REGION Network 40: MGF BACKWASH INLET VALVE ABFV-103 OPEN COMMOND FAIL
   RUNG wire#powerrail
      Contact( "FLUSH DB"."ABFV 103 MULTIGRADE FILTER VALVE" )
      wire#w1
      Coil( "ALARM DB"."MGF BACKWASH INLET VALVE ABFV-103 OPEN COMMOND FAIL" )
   END_RUNG
   RUNG wire#w1
      P_Trig( "P_TRIG".ARR[39] )
      S_Coil( "OUTPUT MAPPING DB"."HOOTER RESET" )
   END_RUNG
   // the same network as SCL:
   "ALARM DB"."MGF BACKWASH INLET VALVE ABFV-103 OPEN COMMOND FAIL" := "FLUSH DB"."ABFV 103 MULTIGRADE FILTER VALVE";
   #_w1 := "FLUSH DB"."ABFV 103 MULTIGRADE FILTER VALVE" AND NOT "P_TRIG".ARR[39];   // rising edge
   "P_TRIG".ARR[39] := "FLUSH DB"."ABFV 103 MULTIGRADE FILTER VALVE";
   IF #_w1 THEN "OUTPUT MAPPING DB"."HOOTER RESET" := TRUE; END_IF;
END_REGION

REGION Network 41: MGF BACKWASH INLET VALVE ABFV-103 CLOSE COMMOND FAIL
   RUNG wire#powerrail
      Contact( "FLUSH DB"."ABFV 103 MULTIGRADE FILTER VALVE_CLOSE" )
      wire#w1
      Coil( "ALARM DB"."MGF BACKWASH INLET VALVE ABFV-103 CLOSE COMMOND FAIL" )
   END_RUNG
   RUNG wire#w1
      P_Trig( "P_TRIG".ARR[40] )
      S_Coil( "OUTPUT MAPPING DB"."HOOTER RESET" )
   END_RUNG
   // the same network as SCL:
   "ALARM DB"."MGF BACKWASH INLET VALVE ABFV-103 CLOSE COMMOND FAIL" := "FLUSH DB"."ABFV 103 MULTIGRADE FILTER VALVE_CLOSE";
   #_w1 := "FLUSH DB"."ABFV 103 MULTIGRADE FILTER VALVE_CLOSE" AND NOT "P_TRIG".ARR[40];   // rising edge
   "P_TRIG".ARR[40] := "FLUSH DB"."ABFV 103 MULTIGRADE FILTER VALVE_CLOSE";
   IF #_w1 THEN "OUTPUT MAPPING DB"."HOOTER RESET" := TRUE; END_IF;
END_REGION

REGION Network 42: MGF OUTLET VALVE ABFV-104 OPEN COMMOND FAIL
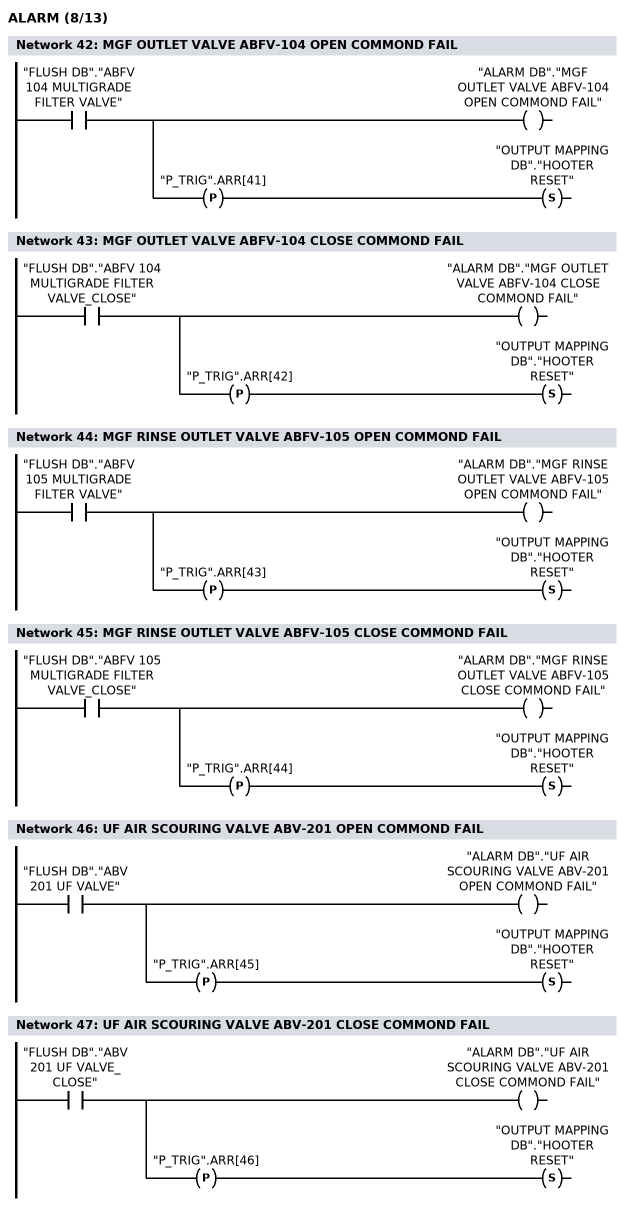
   RUNG wire#powerrail
      Contact( "FLUSH DB"."ABFV 104 MULTIGRADE FILTER VALVE" )
      wire#w1
      Coil( "ALARM DB"."MGF OUTLET VALVE ABFV-104 OPEN COMMOND FAIL" )
   END_RUNG
   RUNG wire#w1
      P_Trig( "P_TRIG".ARR[41] )
      S_Coil( "OUTPUT MAPPING DB"."HOOTER RESET" )
   END_RUNG
   // the same network as SCL:
   "ALARM DB"."MGF OUTLET VALVE ABFV-104 OPEN COMMOND FAIL" := "FLUSH DB"."ABFV 104 MULTIGRADE FILTER VALVE";
   #_w1 := "FLUSH DB"."ABFV 104 MULTIGRADE FILTER VALVE" AND NOT "P_TRIG".ARR[41];   // rising edge
   "P_TRIG".ARR[41] := "FLUSH DB"."ABFV 104 MULTIGRADE FILTER VALVE";
   IF #_w1 THEN "OUTPUT MAPPING DB"."HOOTER RESET" := TRUE; END_IF;
END_REGION

REGION Network 43: MGF OUTLET VALVE ABFV-104 CLOSE COMMOND FAIL
   RUNG wire#powerrail
      Contact( "FLUSH DB"."ABFV 104 MULTIGRADE FILTER VALVE_CLOSE" )
      wire#w1
      Coil( "ALARM DB"."MGF OUTLET VALVE ABFV-104 CLOSE COMMOND FAIL" )
   END_RUNG
   RUNG wire#w1
      P_Trig( "P_TRIG".ARR[42] )
      S_Coil( "OUTPUT MAPPING DB"."HOOTER RESET" )
   END_RUNG
   // the same network as SCL:
   "ALARM DB"."MGF OUTLET VALVE ABFV-104 CLOSE COMMOND FAIL" := "FLUSH DB"."ABFV 104 MULTIGRADE FILTER VALVE_CLOSE";
   #_w1 := "FLUSH DB"."ABFV 104 MULTIGRADE FILTER VALVE_CLOSE" AND NOT "P_TRIG".ARR[42];   // rising edge
   "P_TRIG".ARR[42] := "FLUSH DB"."ABFV 104 MULTIGRADE FILTER VALVE_CLOSE";
   IF #_w1 THEN "OUTPUT MAPPING DB"."HOOTER RESET" := TRUE; END_IF;
END_REGION

REGION Network 44: MGF RINSE OUTLET VALVE ABFV-105 OPEN COMMOND FAIL
   RUNG wire#powerrail
      Contact( "FLUSH DB"."ABFV 105 MULTIGRADE FILTER VALVE" )
      wire#w1
      Coil( "ALARM DB"."MGF RINSE OUTLET VALVE ABFV-105 OPEN COMMOND FAIL" )
   END_RUNG
   RUNG wire#w1
      P_Trig( "P_TRIG".ARR[43] )
      S_Coil( "OUTPUT MAPPING DB"."HOOTER RESET" )
   END_RUNG
   // the same network as SCL:
   "ALARM DB"."MGF RINSE OUTLET VALVE ABFV-105 OPEN COMMOND FAIL" := "FLUSH DB"."ABFV 105 MULTIGRADE FILTER VALVE";
   #_w1 := "FLUSH DB"."ABFV 105 MULTIGRADE FILTER VALVE" AND NOT "P_TRIG".ARR[43];   // rising edge
   "P_TRIG".ARR[43] := "FLUSH DB"."ABFV 105 MULTIGRADE FILTER VALVE";
   IF #_w1 THEN "OUTPUT MAPPING DB"."HOOTER RESET" := TRUE; END_IF;
END_REGION

REGION Network 45: MGF RINSE OUTLET VALVE ABFV-105 CLOSE COMMOND FAIL
   RUNG wire#powerrail
      Contact( "FLUSH DB"."ABFV 105 MULTIGRADE FILTER VALVE_CLOSE" )
      wire#w1
      Coil( "ALARM DB"."MGF RINSE OUTLET VALVE ABFV-105 CLOSE COMMOND FAIL" )
   END_RUNG
   RUNG wire#w1
      P_Trig( "P_TRIG".ARR[44] )
      S_Coil( "OUTPUT MAPPING DB"."HOOTER RESET" )
   END_RUNG
   // the same network as SCL:
   "ALARM DB"."MGF RINSE OUTLET VALVE ABFV-105 CLOSE COMMOND FAIL" := "FLUSH DB"."ABFV 105 MULTIGRADE FILTER VALVE_CLOSE";
   #_w1 := "FLUSH DB"."ABFV 105 MULTIGRADE FILTER VALVE_CLOSE" AND NOT "P_TRIG".ARR[44];   // rising edge
   "P_TRIG".ARR[44] := "FLUSH DB"."ABFV 105 MULTIGRADE FILTER VALVE_CLOSE";
   IF #_w1 THEN "OUTPUT MAPPING DB"."HOOTER RESET" := TRUE; END_IF;
END_REGION

REGION Network 46: UF AIR SCOURING VALVE ABV-201 OPEN COMMOND FAIL
   RUNG wire#powerrail
      Contact( "FLUSH DB"."ABV 201 UF VALVE" )
      wire#w1
      Coil( "ALARM DB"."UF AIR SCOURING VALVE ABV-201 OPEN COMMOND FAIL" )
   END_RUNG
   RUNG wire#w1
      P_Trig( "P_TRIG".ARR[45] )
      S_Coil( "OUTPUT MAPPING DB"."HOOTER RESET" )
   END_RUNG
   // the same network as SCL:
   "ALARM DB"."UF AIR SCOURING VALVE ABV-201 OPEN COMMOND FAIL" := "FLUSH DB"."ABV 201 UF VALVE";
   #_w1 := "FLUSH DB"."ABV 201 UF VALVE" AND NOT "P_TRIG".ARR[45];   // rising edge
   "P_TRIG".ARR[45] := "FLUSH DB"."ABV 201 UF VALVE";
   IF #_w1 THEN "OUTPUT MAPPING DB"."HOOTER RESET" := TRUE; END_IF;
END_REGION

REGION Network 47: UF AIR SCOURING VALVE ABV-201 CLOSE COMMOND FAIL
   RUNG wire#powerrail
      Contact( "FLUSH DB"."ABV 201 UF VALVE_CLOSE" )
      wire#w1
      Coil( "ALARM DB"."UF AIR SCOURING VALVE ABV-201 CLOSE COMMOND FAIL" )
   END_RUNG
   RUNG wire#w1
      P_Trig( "P_TRIG".ARR[46] )
      S_Coil( "OUTPUT MAPPING DB"."HOOTER RESET" )
   END_RUNG
   // the same network as SCL:
   "ALARM DB"."UF AIR SCOURING VALVE ABV-201 CLOSE COMMOND FAIL" := "FLUSH DB"."ABV 201 UF VALVE_CLOSE";
   #_w1 := "FLUSH DB"."ABV 201 UF VALVE_CLOSE" AND NOT "P_TRIG".ARR[46];   // rising edge
   "P_TRIG".ARR[46] := "FLUSH DB"."ABV 201 UF VALVE_CLOSE";
   IF #_w1 THEN "OUTPUT MAPPING DB"."HOOTER RESET" := TRUE; END_IF;
END_REGION

REGION Network 48: UF INLET VALVE ABFV-201 OPEN COMMOND FAIL
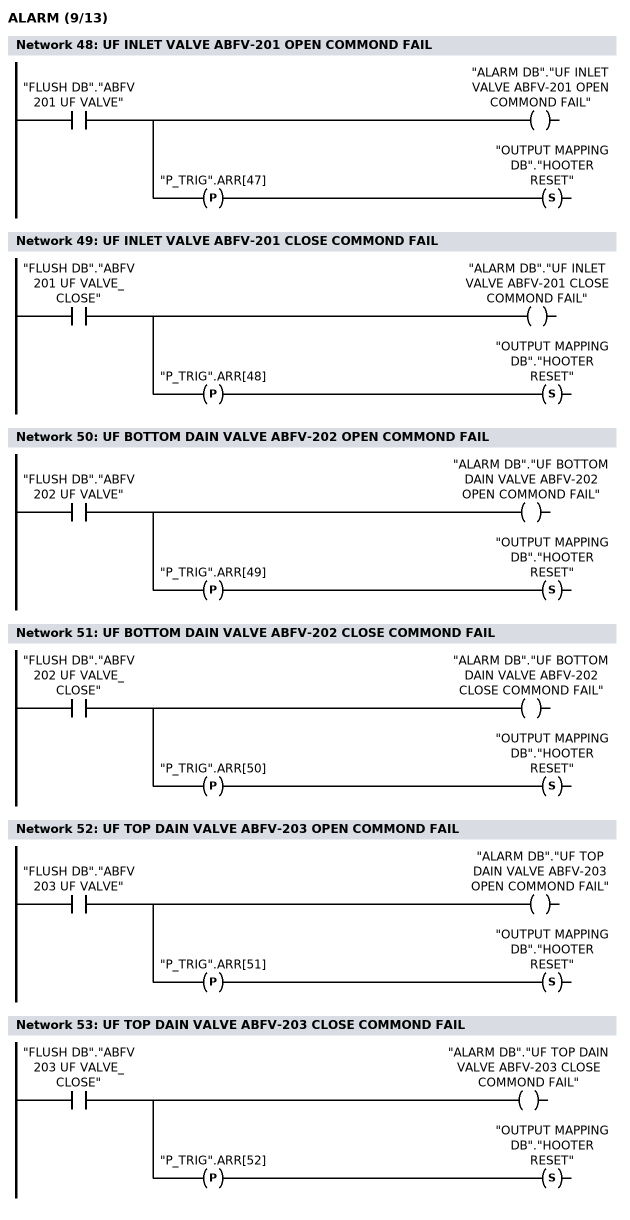
   RUNG wire#powerrail
      Contact( "FLUSH DB"."ABFV 201 UF VALVE" )
      wire#w1
      Coil( "ALARM DB"."UF INLET VALVE ABFV-201 OPEN COMMOND FAIL" )
   END_RUNG
   RUNG wire#w1
      P_Trig( "P_TRIG".ARR[47] )
      S_Coil( "OUTPUT MAPPING DB"."HOOTER RESET" )
   END_RUNG
   // the same network as SCL:
   "ALARM DB"."UF INLET VALVE ABFV-201 OPEN COMMOND FAIL" := "FLUSH DB"."ABFV 201 UF VALVE";
   #_w1 := "FLUSH DB"."ABFV 201 UF VALVE" AND NOT "P_TRIG".ARR[47];   // rising edge
   "P_TRIG".ARR[47] := "FLUSH DB"."ABFV 201 UF VALVE";
   IF #_w1 THEN "OUTPUT MAPPING DB"."HOOTER RESET" := TRUE; END_IF;
END_REGION

REGION Network 49: UF INLET VALVE ABFV-201 CLOSE COMMOND FAIL
   RUNG wire#powerrail
      Contact( "FLUSH DB"."ABFV 201 UF VALVE_CLOSE" )
      wire#w1
      Coil( "ALARM DB"."UF INLET VALVE ABFV-201 CLOSE COMMOND FAIL" )
   END_RUNG
   RUNG wire#w1
      P_Trig( "P_TRIG".ARR[48] )
      S_Coil( "OUTPUT MAPPING DB"."HOOTER RESET" )
   END_RUNG
   // the same network as SCL:
   "ALARM DB"."UF INLET VALVE ABFV-201 CLOSE COMMOND FAIL" := "FLUSH DB"."ABFV 201 UF VALVE_CLOSE";
   #_w1 := "FLUSH DB"."ABFV 201 UF VALVE_CLOSE" AND NOT "P_TRIG".ARR[48];   // rising edge
   "P_TRIG".ARR[48] := "FLUSH DB"."ABFV 201 UF VALVE_CLOSE";
   IF #_w1 THEN "OUTPUT MAPPING DB"."HOOTER RESET" := TRUE; END_IF;
END_REGION

REGION Network 50: UF BOTTOM DAIN VALVE ABFV-202 OPEN COMMOND FAIL
   RUNG wire#powerrail
      Contact( "FLUSH DB"."ABFV 202 UF VALVE" )
      wire#w1
      Coil( "ALARM DB"."UF BOTTOM DAIN VALVE ABFV-202 OPEN COMMOND FAIL" )
   END_RUNG
   RUNG wire#w1
      P_Trig( "P_TRIG".ARR[49] )
      S_Coil( "OUTPUT MAPPING DB"."HOOTER RESET" )
   END_RUNG
   // the same network as SCL:
   "ALARM DB"."UF BOTTOM DAIN VALVE ABFV-202 OPEN COMMOND FAIL" := "FLUSH DB"."ABFV 202 UF VALVE";
   #_w1 := "FLUSH DB"."ABFV 202 UF VALVE" AND NOT "P_TRIG".ARR[49];   // rising edge
   "P_TRIG".ARR[49] := "FLUSH DB"."ABFV 202 UF VALVE";
   IF #_w1 THEN "OUTPUT MAPPING DB"."HOOTER RESET" := TRUE; END_IF;
END_REGION

REGION Network 51: UF BOTTOM DAIN VALVE ABFV-202 CLOSE COMMOND FAIL
   RUNG wire#powerrail
      Contact( "FLUSH DB"."ABFV 202 UF VALVE_CLOSE" )
      wire#w1
      Coil( "ALARM DB"."UF BOTTOM DAIN VALVE ABFV-202 CLOSE COMMOND FAIL" )
   END_RUNG
   RUNG wire#w1
      P_Trig( "P_TRIG".ARR[50] )
      S_Coil( "OUTPUT MAPPING DB"."HOOTER RESET" )
   END_RUNG
   // the same network as SCL:
   "ALARM DB"."UF BOTTOM DAIN VALVE ABFV-202 CLOSE COMMOND FAIL" := "FLUSH DB"."ABFV 202 UF VALVE_CLOSE";
   #_w1 := "FLUSH DB"."ABFV 202 UF VALVE_CLOSE" AND NOT "P_TRIG".ARR[50];   // rising edge
   "P_TRIG".ARR[50] := "FLUSH DB"."ABFV 202 UF VALVE_CLOSE";
   IF #_w1 THEN "OUTPUT MAPPING DB"."HOOTER RESET" := TRUE; END_IF;
END_REGION

REGION Network 52: UF TOP DAIN VALVE ABFV-203 OPEN COMMOND FAIL
   RUNG wire#powerrail
      Contact( "FLUSH DB"."ABFV 203 UF VALVE" )
      wire#w1
      Coil( "ALARM DB"."UF TOP DAIN VALVE ABFV-203 OPEN COMMOND FAIL" )
   END_RUNG
   RUNG wire#w1
      P_Trig( "P_TRIG".ARR[51] )
      S_Coil( "OUTPUT MAPPING DB"."HOOTER RESET" )
   END_RUNG
   // the same network as SCL:
   "ALARM DB"."UF TOP DAIN VALVE ABFV-203 OPEN COMMOND FAIL" := "FLUSH DB"."ABFV 203 UF VALVE";
   #_w1 := "FLUSH DB"."ABFV 203 UF VALVE" AND NOT "P_TRIG".ARR[51];   // rising edge
   "P_TRIG".ARR[51] := "FLUSH DB"."ABFV 203 UF VALVE";
   IF #_w1 THEN "OUTPUT MAPPING DB"."HOOTER RESET" := TRUE; END_IF;
END_REGION

REGION Network 53: UF TOP DAIN VALVE ABFV-203 CLOSE COMMOND FAIL
   RUNG wire#powerrail
      Contact( "FLUSH DB"."ABFV 203 UF VALVE_CLOSE" )
      wire#w1
      Coil( "ALARM DB"."UF TOP DAIN VALVE ABFV-203 CLOSE COMMOND FAIL" )
   END_RUNG
   RUNG wire#w1
      P_Trig( "P_TRIG".ARR[52] )
      S_Coil( "OUTPUT MAPPING DB"."HOOTER RESET" )
   END_RUNG
   // the same network as SCL:
   "ALARM DB"."UF TOP DAIN VALVE ABFV-203 CLOSE COMMOND FAIL" := "FLUSH DB"."ABFV 203 UF VALVE_CLOSE";
   #_w1 := "FLUSH DB"."ABFV 203 UF VALVE_CLOSE" AND NOT "P_TRIG".ARR[52];   // rising edge
   "P_TRIG".ARR[52] := "FLUSH DB"."ABFV 203 UF VALVE_CLOSE";
   IF #_w1 THEN "OUTPUT MAPPING DB"."HOOTER RESET" := TRUE; END_IF;
END_REGION

REGION Network 54: UF BACKWASH INLET VALVE ABFV-204 OPEN COMMOND FAIL
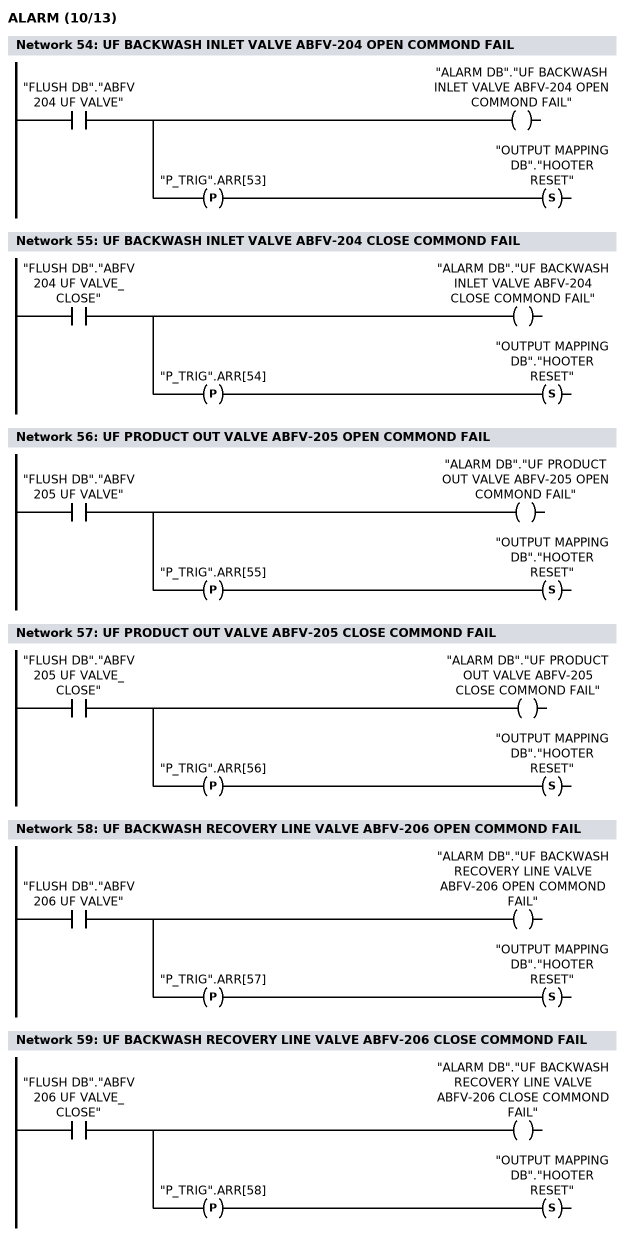
   RUNG wire#powerrail
      Contact( "FLUSH DB"."ABFV 204 UF VALVE" )
      wire#w1
      Coil( "ALARM DB"."UF BACKWASH INLET VALVE ABFV-204 OPEN COMMOND FAIL" )
   END_RUNG
   RUNG wire#w1
      P_Trig( "P_TRIG".ARR[53] )
      S_Coil( "OUTPUT MAPPING DB"."HOOTER RESET" )
   END_RUNG
   // the same network as SCL:
   "ALARM DB"."UF BACKWASH INLET VALVE ABFV-204 OPEN COMMOND FAIL" := "FLUSH DB"."ABFV 204 UF VALVE";
   #_w1 := "FLUSH DB"."ABFV 204 UF VALVE" AND NOT "P_TRIG".ARR[53];   // rising edge
   "P_TRIG".ARR[53] := "FLUSH DB"."ABFV 204 UF VALVE";
   IF #_w1 THEN "OUTPUT MAPPING DB"."HOOTER RESET" := TRUE; END_IF;
END_REGION

REGION Network 55: UF BACKWASH INLET VALVE ABFV-204 CLOSE COMMOND FAIL
   RUNG wire#powerrail
      Contact( "FLUSH DB"."ABFV 204 UF VALVE_CLOSE" )
      wire#w1
      Coil( "ALARM DB"."UF BACKWASH INLET VALVE ABFV-204 CLOSE COMMOND FAIL" )
   END_RUNG
   RUNG wire#w1
      P_Trig( "P_TRIG".ARR[54] )
      S_Coil( "OUTPUT MAPPING DB"."HOOTER RESET" )
   END_RUNG
   // the same network as SCL:
   "ALARM DB"."UF BACKWASH INLET VALVE ABFV-204 CLOSE COMMOND FAIL" := "FLUSH DB"."ABFV 204 UF VALVE_CLOSE";
   #_w1 := "FLUSH DB"."ABFV 204 UF VALVE_CLOSE" AND NOT "P_TRIG".ARR[54];   // rising edge
   "P_TRIG".ARR[54] := "FLUSH DB"."ABFV 204 UF VALVE_CLOSE";
   IF #_w1 THEN "OUTPUT MAPPING DB"."HOOTER RESET" := TRUE; END_IF;
END_REGION

REGION Network 56: UF PRODUCT OUT VALVE ABFV-205 OPEN COMMOND FAIL
   RUNG wire#powerrail
      Contact( "FLUSH DB"."ABFV 205 UF VALVE" )
      wire#w1
      Coil( "ALARM DB"."UF PRODUCT OUT VALVE ABFV-205 OPEN COMMOND FAIL" )
   END_RUNG
   RUNG wire#w1
      P_Trig( "P_TRIG".ARR[55] )
      S_Coil( "OUTPUT MAPPING DB"."HOOTER RESET" )
   END_RUNG
   // the same network as SCL:
   "ALARM DB"."UF PRODUCT OUT VALVE ABFV-205 OPEN COMMOND FAIL" := "FLUSH DB"."ABFV 205 UF VALVE";
   #_w1 := "FLUSH DB"."ABFV 205 UF VALVE" AND NOT "P_TRIG".ARR[55];   // rising edge
   "P_TRIG".ARR[55] := "FLUSH DB"."ABFV 205 UF VALVE";
   IF #_w1 THEN "OUTPUT MAPPING DB"."HOOTER RESET" := TRUE; END_IF;
END_REGION

REGION Network 57: UF PRODUCT OUT VALVE ABFV-205 CLOSE COMMOND FAIL
   RUNG wire#powerrail
      Contact( "FLUSH DB"."ABFV 205 UF VALVE_CLOSE" )
      wire#w1
      Coil( "ALARM DB"."UF PRODUCT OUT VALVE ABFV-205 CLOSE COMMOND FAIL" )
   END_RUNG
   RUNG wire#w1
      P_Trig( "P_TRIG".ARR[56] )
      S_Coil( "OUTPUT MAPPING DB"."HOOTER RESET" )
   END_RUNG
   // the same network as SCL:
   "ALARM DB"."UF PRODUCT OUT VALVE ABFV-205 CLOSE COMMOND FAIL" := "FLUSH DB"."ABFV 205 UF VALVE_CLOSE";
   #_w1 := "FLUSH DB"."ABFV 205 UF VALVE_CLOSE" AND NOT "P_TRIG".ARR[56];   // rising edge
   "P_TRIG".ARR[56] := "FLUSH DB"."ABFV 205 UF VALVE_CLOSE";
   IF #_w1 THEN "OUTPUT MAPPING DB"."HOOTER RESET" := TRUE; END_IF;
END_REGION

REGION Network 58: UF BACKWASH RECOVERY LINE VALVE ABFV-206 OPEN COMMOND FAIL
   RUNG wire#powerrail
      Contact( "FLUSH DB"."ABFV 206 UF VALVE" )
      wire#w1
      Coil( "ALARM DB"."UF BACKWASH RECOVERY LINE VALVE ABFV-206 OPEN COMMOND FAIL" )
   END_RUNG
   RUNG wire#w1
      P_Trig( "P_TRIG".ARR[57] )
      S_Coil( "OUTPUT MAPPING DB"."HOOTER RESET" )
   END_RUNG
   // the same network as SCL:
   "ALARM DB"."UF BACKWASH RECOVERY LINE VALVE ABFV-206 OPEN COMMOND FAIL" := "FLUSH DB"."ABFV 206 UF VALVE";
   #_w1 := "FLUSH DB"."ABFV 206 UF VALVE" AND NOT "P_TRIG".ARR[57];   // rising edge
   "P_TRIG".ARR[57] := "FLUSH DB"."ABFV 206 UF VALVE";
   IF #_w1 THEN "OUTPUT MAPPING DB"."HOOTER RESET" := TRUE; END_IF;
END_REGION

REGION Network 59: UF BACKWASH RECOVERY LINE VALVE ABFV-206 CLOSE COMMOND FAIL
   RUNG wire#powerrail
      Contact( "FLUSH DB"."ABFV 206 UF VALVE_CLOSE" )
      wire#w1
      Coil( "ALARM DB"."UF BACKWASH RECOVERY LINE VALVE ABFV-206 CLOSE COMMOND FAIL" )
   END_RUNG
   RUNG wire#w1
      P_Trig( "P_TRIG".ARR[58] )
      S_Coil( "OUTPUT MAPPING DB"."HOOTER RESET" )
   END_RUNG
   // the same network as SCL:
   "ALARM DB"."UF BACKWASH RECOVERY LINE VALVE ABFV-206 CLOSE COMMOND FAIL" := "FLUSH DB"."ABFV 206 UF VALVE_CLOSE";
   #_w1 := "FLUSH DB"."ABFV 206 UF VALVE_CLOSE" AND NOT "P_TRIG".ARR[58];   // rising edge
   "P_TRIG".ARR[58] := "FLUSH DB"."ABFV 206 UF VALVE_CLOSE";
   IF #_w1 THEN "OUTPUT MAPPING DB"."HOOTER RESET" := TRUE; END_IF;
END_REGION

REGION Network 60: UF BACKWASH DRAIN LINE VALVE ABFV-207 OPEN COMMOND FAIL
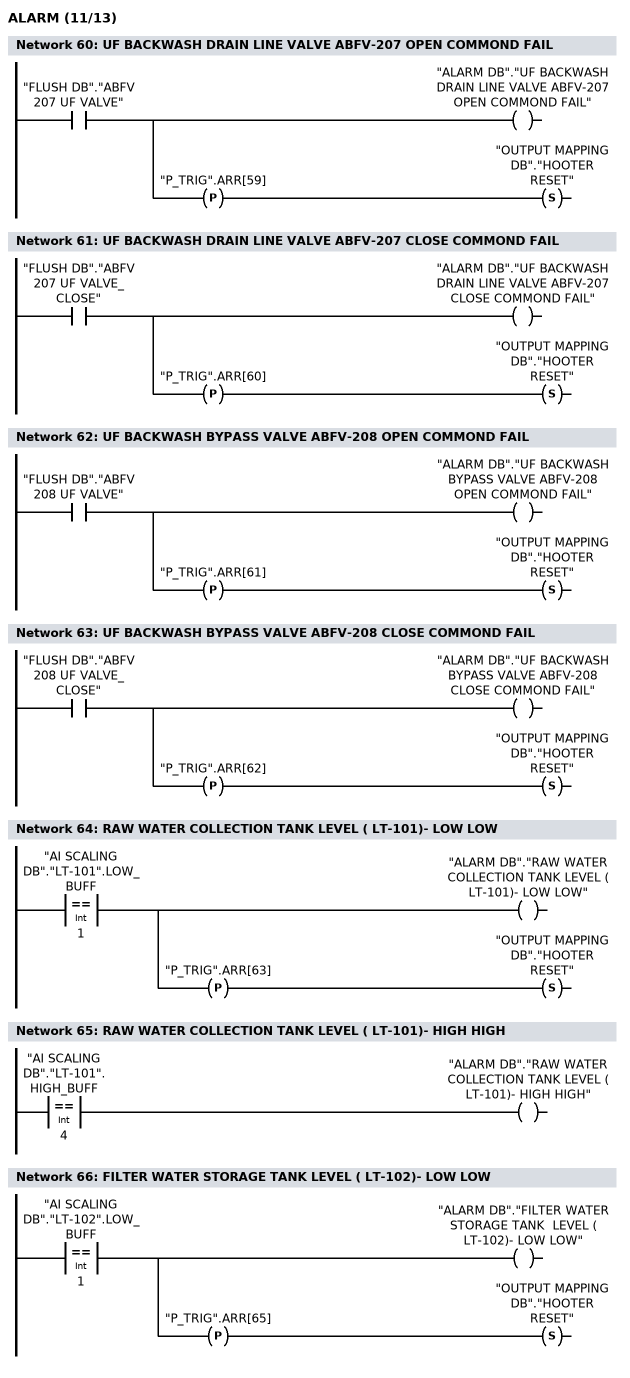
   RUNG wire#powerrail
      Contact( "FLUSH DB"."ABFV 207 UF VALVE" )
      wire#w1
      Coil( "ALARM DB"."UF BACKWASH DRAIN LINE VALVE ABFV-207 OPEN COMMOND FAIL" )
   END_RUNG
   RUNG wire#w1
      P_Trig( "P_TRIG".ARR[59] )
      S_Coil( "OUTPUT MAPPING DB"."HOOTER RESET" )
   END_RUNG
   // the same network as SCL:
   "ALARM DB"."UF BACKWASH DRAIN LINE VALVE ABFV-207 OPEN COMMOND FAIL" := "FLUSH DB"."ABFV 207 UF VALVE";
   #_w1 := "FLUSH DB"."ABFV 207 UF VALVE" AND NOT "P_TRIG".ARR[59];   // rising edge
   "P_TRIG".ARR[59] := "FLUSH DB"."ABFV 207 UF VALVE";
   IF #_w1 THEN "OUTPUT MAPPING DB"."HOOTER RESET" := TRUE; END_IF;
END_REGION

REGION Network 61: UF BACKWASH DRAIN LINE VALVE ABFV-207 CLOSE COMMOND FAIL
   RUNG wire#powerrail
      Contact( "FLUSH DB"."ABFV 207 UF VALVE_CLOSE" )
      wire#w1
      Coil( "ALARM DB"."UF BACKWASH DRAIN LINE VALVE ABFV-207 CLOSE COMMOND FAIL" )
   END_RUNG
   RUNG wire#w1
      P_Trig( "P_TRIG".ARR[60] )
      S_Coil( "OUTPUT MAPPING DB"."HOOTER RESET" )
   END_RUNG
   // the same network as SCL:
   "ALARM DB"."UF BACKWASH DRAIN LINE VALVE ABFV-207 CLOSE COMMOND FAIL" := "FLUSH DB"."ABFV 207 UF VALVE_CLOSE";
   #_w1 := "FLUSH DB"."ABFV 207 UF VALVE_CLOSE" AND NOT "P_TRIG".ARR[60];   // rising edge
   "P_TRIG".ARR[60] := "FLUSH DB"."ABFV 207 UF VALVE_CLOSE";
   IF #_w1 THEN "OUTPUT MAPPING DB"."HOOTER RESET" := TRUE; END_IF;
END_REGION

REGION Network 62: UF BACKWASH BYPASS VALVE ABFV-208 OPEN COMMOND FAIL
   RUNG wire#powerrail
      Contact( "FLUSH DB"."ABFV 208 UF VALVE" )
      wire#w1
      Coil( "ALARM DB"."UF BACKWASH BYPASS VALVE ABFV-208 OPEN COMMOND FAIL" )
   END_RUNG
   RUNG wire#w1
      P_Trig( "P_TRIG".ARR[61] )
      S_Coil( "OUTPUT MAPPING DB"."HOOTER RESET" )
   END_RUNG
   // the same network as SCL:
   "ALARM DB"."UF BACKWASH BYPASS VALVE ABFV-208 OPEN COMMOND FAIL" := "FLUSH DB"."ABFV 208 UF VALVE";
   #_w1 := "FLUSH DB"."ABFV 208 UF VALVE" AND NOT "P_TRIG".ARR[61];   // rising edge
   "P_TRIG".ARR[61] := "FLUSH DB"."ABFV 208 UF VALVE";
   IF #_w1 THEN "OUTPUT MAPPING DB"."HOOTER RESET" := TRUE; END_IF;
END_REGION

REGION Network 63: UF BACKWASH BYPASS VALVE ABFV-208 CLOSE COMMOND FAIL
   RUNG wire#powerrail
      Contact( "FLUSH DB"."ABFV 208 UF VALVE_CLOSE" )
      wire#w1
      Coil( "ALARM DB"."UF BACKWASH BYPASS VALVE ABFV-208 CLOSE COMMOND FAIL" )
   END_RUNG
   RUNG wire#w1
      P_Trig( "P_TRIG".ARR[62] )
      S_Coil( "OUTPUT MAPPING DB"."HOOTER RESET" )
   END_RUNG
   // the same network as SCL:
   "ALARM DB"."UF BACKWASH BYPASS VALVE ABFV-208 CLOSE COMMOND FAIL" := "FLUSH DB"."ABFV 208 UF VALVE_CLOSE";
   #_w1 := "FLUSH DB"."ABFV 208 UF VALVE_CLOSE" AND NOT "P_TRIG".ARR[62];   // rising edge
   "P_TRIG".ARR[62] := "FLUSH DB"."ABFV 208 UF VALVE_CLOSE";
   IF #_w1 THEN "OUTPUT MAPPING DB"."HOOTER RESET" := TRUE; END_IF;
END_REGION

REGION Network 64: RAW WATER COLLECTION TANK LEVEL ( LT-101)- LOW LOW
   RUNG wire#powerrail
      { S7_Templates := "SrcType := Int" } EQ_Contact(in1 := "AI SCALING DB"."LT-101".LOW_BUFF, in2 := 1)
      wire#w1
      Coil( "ALARM DB"."RAW WATER COLLECTION TANK LEVEL ( LT-101)- LOW LOW" )
   END_RUNG
   RUNG wire#w1
      P_Trig( "P_TRIG".ARR[63] )
      S_Coil( "OUTPUT MAPPING DB"."HOOTER RESET" )
   END_RUNG
   // the same network as SCL:
   "ALARM DB"."RAW WATER COLLECTION TANK LEVEL ( LT-101)- LOW LOW" := "AI SCALING DB"."LT-101".LOW_BUFF = 1;
   #_w1 := "ALARM DB"."RAW WATER COLLECTION TANK LEVEL ( LT-101)- LOW LOW" AND NOT "P_TRIG".ARR[63];   // rising edge
   "P_TRIG".ARR[63] := "ALARM DB"."RAW WATER COLLECTION TANK LEVEL ( LT-101)- LOW LOW";
   IF #_w1 THEN "OUTPUT MAPPING DB"."HOOTER RESET" := TRUE; END_IF;
END_REGION

REGION Network 65: RAW WATER COLLECTION TANK LEVEL ( LT-101)- HIGH HIGH
   RUNG wire#powerrail
      { S7_Templates := "SrcType := Int" } EQ_Contact(in1 := "AI SCALING DB"."LT-101".HIGH_BUFF, in2 := 4)
      Coil( "ALARM DB"."RAW WATER COLLECTION TANK LEVEL ( LT-101)- HIGH HIGH" )
   END_RUNG
   // the same network as SCL:
   "ALARM DB"."RAW WATER COLLECTION TANK LEVEL ( LT-101)- HIGH HIGH" := "AI SCALING DB"."LT-101".HIGH_BUFF = 4;
END_REGION

REGION Network 66: FILTER WATER STORAGE TANK LEVEL ( LT-102)- LOW LOW
   RUNG wire#powerrail
      { S7_Templates := "SrcType := Int" } EQ_Contact(in1 := "AI SCALING DB"."LT-102".LOW_BUFF, in2 := 1)
      wire#w1
      Coil( "ALARM DB"."FILTER WATER STORAGE TANK  LEVEL ( LT-102)- LOW LOW" )
   END_RUNG
   RUNG wire#w1
      P_Trig( "P_TRIG".ARR[65] )
      S_Coil( "OUTPUT MAPPING DB"."HOOTER RESET" )
   END_RUNG
   // the same network as SCL:
   "ALARM DB"."FILTER WATER STORAGE TANK  LEVEL ( LT-102)- LOW LOW" := "AI SCALING DB"."LT-102".LOW_BUFF = 1;
   #_w1 := "ALARM DB"."FILTER WATER STORAGE TANK  LEVEL ( LT-102)- LOW LOW" AND NOT "P_TRIG".ARR[65];   // rising edge
   "P_TRIG".ARR[65] := "ALARM DB"."FILTER WATER STORAGE TANK  LEVEL ( LT-102)- LOW LOW";
   IF #_w1 THEN "OUTPUT MAPPING DB"."HOOTER RESET" := TRUE; END_IF;
END_REGION

REGION Network 67: FILTER WATER STORAGE TANK LEVEL ( LT-102)- HIGH HIGH
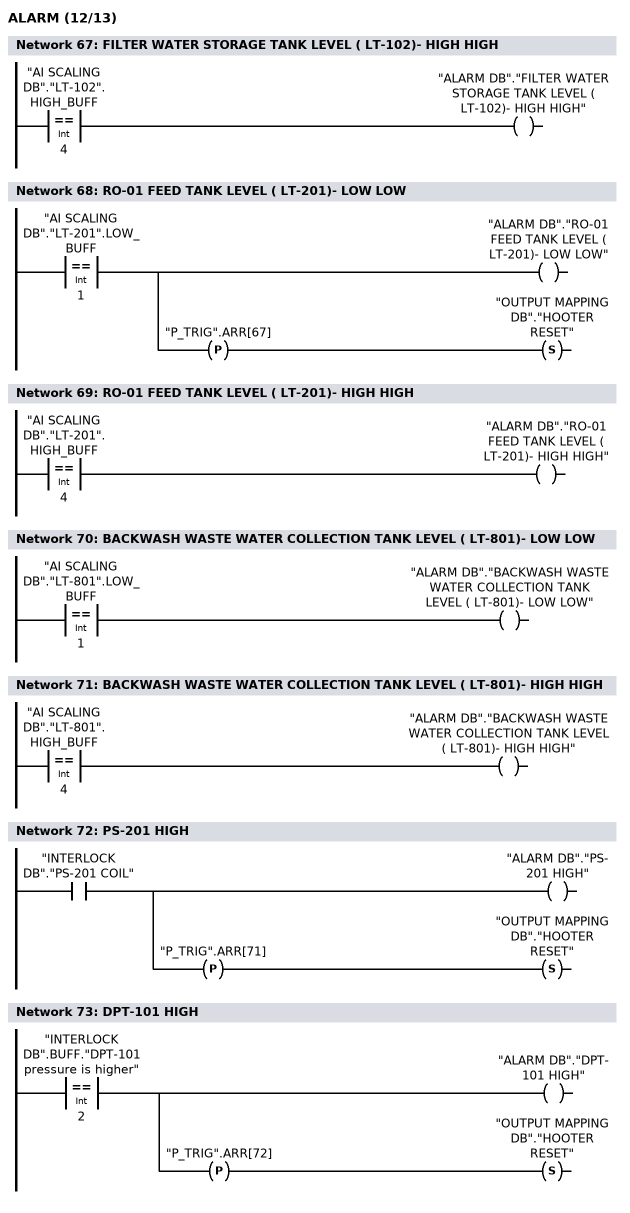
   RUNG wire#powerrail
      { S7_Templates := "SrcType := Int" } EQ_Contact(in1 := "AI SCALING DB"."LT-102".HIGH_BUFF, in2 := 4)
      Coil( "ALARM DB"."FILTER WATER STORAGE TANK LEVEL ( LT-102)- HIGH HIGH" )
   END_RUNG
   // the same network as SCL:
   "ALARM DB"."FILTER WATER STORAGE TANK LEVEL ( LT-102)- HIGH HIGH" := "AI SCALING DB"."LT-102".HIGH_BUFF = 4;
END_REGION

REGION Network 68: RO-01 FEED TANK LEVEL ( LT-201)- LOW LOW
   RUNG wire#powerrail
      { S7_Templates := "SrcType := Int" } EQ_Contact(in1 := "AI SCALING DB"."LT-201".LOW_BUFF, in2 := 1)
      wire#w1
      Coil( "ALARM DB"."RO-01 FEED TANK LEVEL ( LT-201)- LOW LOW" )
   END_RUNG
   RUNG wire#w1
      P_Trig( "P_TRIG".ARR[67] )
      S_Coil( "OUTPUT MAPPING DB"."HOOTER RESET" )
   END_RUNG
   // the same network as SCL:
   "ALARM DB"."RO-01 FEED TANK LEVEL ( LT-201)- LOW LOW" := "AI SCALING DB"."LT-201".LOW_BUFF = 1;
   #_w1 := "ALARM DB"."RO-01 FEED TANK LEVEL ( LT-201)- LOW LOW" AND NOT "P_TRIG".ARR[67];   // rising edge
   "P_TRIG".ARR[67] := "ALARM DB"."RO-01 FEED TANK LEVEL ( LT-201)- LOW LOW";
   IF #_w1 THEN "OUTPUT MAPPING DB"."HOOTER RESET" := TRUE; END_IF;
END_REGION

REGION Network 69: RO-01 FEED TANK LEVEL ( LT-201)- HIGH HIGH
   RUNG wire#powerrail
      { S7_Templates := "SrcType := Int" } EQ_Contact(in1 := "AI SCALING DB"."LT-201".HIGH_BUFF, in2 := 4)
      Coil( "ALARM DB"."RO-01 FEED TANK LEVEL ( LT-201)- HIGH HIGH" )
   END_RUNG
   // the same network as SCL:
   "ALARM DB"."RO-01 FEED TANK LEVEL ( LT-201)- HIGH HIGH" := "AI SCALING DB"."LT-201".HIGH_BUFF = 4;
END_REGION

REGION Network 70: BACKWASH WASTE WATER COLLECTION TANK LEVEL ( LT-801)- LOW LOW
   RUNG wire#powerrail
      { S7_Templates := "SrcType := Int" } EQ_Contact(in1 := "AI SCALING DB"."LT-801".LOW_BUFF, in2 := 1)
      Coil( "ALARM DB"."BACKWASH WASTE WATER COLLECTION TANK  LEVEL ( LT-801)- LOW LOW" )
   END_RUNG
   // the same network as SCL:
   "ALARM DB"."BACKWASH WASTE WATER COLLECTION TANK  LEVEL ( LT-801)- LOW LOW" := "AI SCALING DB"."LT-801".LOW_BUFF = 1;
END_REGION

REGION Network 71: BACKWASH WASTE WATER COLLECTION TANK LEVEL ( LT-801)- HIGH HIGH
   RUNG wire#powerrail
      { S7_Templates := "SrcType := Int" } EQ_Contact(in1 := "AI SCALING DB"."LT-801".HIGH_BUFF, in2 := 4)
      Coil( "ALARM DB"."BACKWASH WASTE WATER COLLECTION TANK LEVEL ( LT-801)- HIGH HIGH" )
   END_RUNG
   // the same network as SCL:
   "ALARM DB"."BACKWASH WASTE WATER COLLECTION TANK LEVEL ( LT-801)- HIGH HIGH" := "AI SCALING DB"."LT-801".HIGH_BUFF = 4;
END_REGION

REGION Network 72: PS-201 HIGH
   RUNG wire#powerrail
      Contact( "INTERLOCK DB"."PS-201 COIL" )
      wire#w1
      Coil( "ALARM DB"."PS-201 HIGH" )
   END_RUNG
   RUNG wire#w1
      P_Trig( "P_TRIG".ARR[71] )
      S_Coil( "OUTPUT MAPPING DB"."HOOTER RESET" )
   END_RUNG
   // the same network as SCL:
   "ALARM DB"."PS-201 HIGH" := "INTERLOCK DB"."PS-201 COIL";
   #_w1 := "INTERLOCK DB"."PS-201 COIL" AND NOT "P_TRIG".ARR[71];   // rising edge
   "P_TRIG".ARR[71] := "INTERLOCK DB"."PS-201 COIL";
   IF #_w1 THEN "OUTPUT MAPPING DB"."HOOTER RESET" := TRUE; END_IF;
END_REGION

REGION Network 73: DPT-101 HIGH
   RUNG wire#powerrail
      { S7_Templates := "SrcType := Int" } EQ_Contact(in1 := "INTERLOCK DB".BUFF."DPT-101 pressure is higher", in2 := 2)
      wire#w1
      Coil( "ALARM DB"."DPT-101 HIGH" )
   END_RUNG
   RUNG wire#w1
      P_Trig( "P_TRIG".ARR[72] )
      S_Coil( "OUTPUT MAPPING DB"."HOOTER RESET" )
   END_RUNG
   // the same network as SCL:
   "ALARM DB"."DPT-101 HIGH" := "INTERLOCK DB".BUFF."DPT-101 pressure is higher" = 2;
   #_w1 := "ALARM DB"."DPT-101 HIGH" AND NOT "P_TRIG".ARR[72];   // rising edge
   "P_TRIG".ARR[72] := "ALARM DB"."DPT-101 HIGH";
   IF #_w1 THEN "OUTPUT MAPPING DB"."HOOTER RESET" := TRUE; END_IF;
END_REGION

REGION Network 74: DPT-201 HIGH
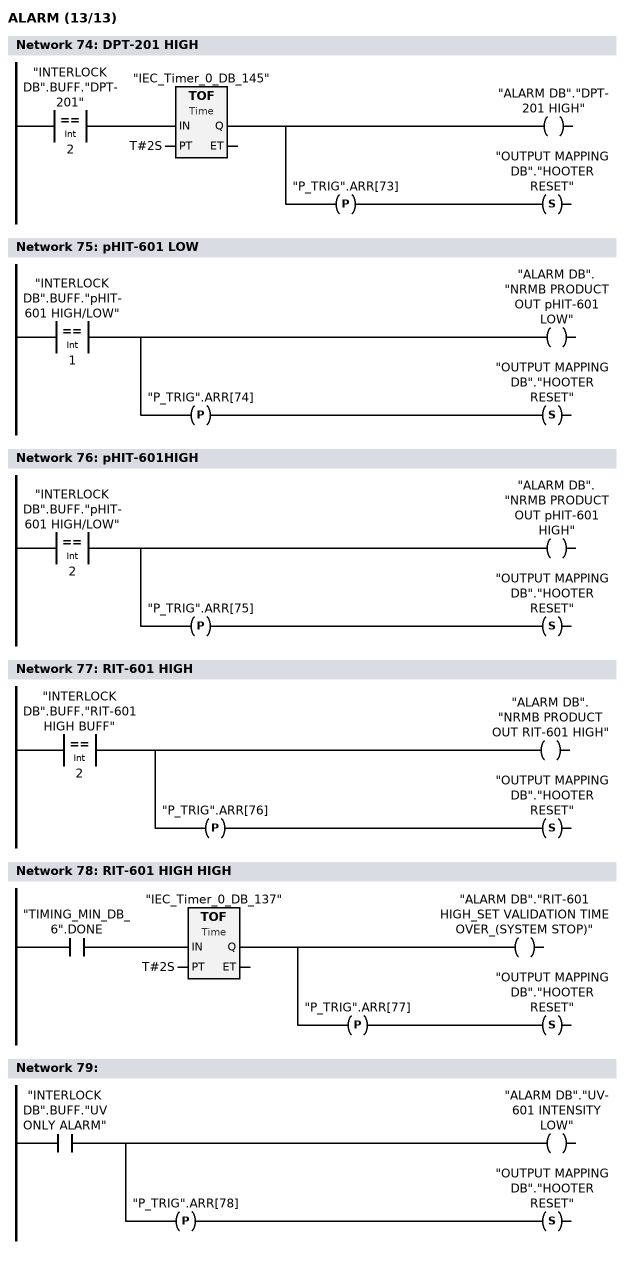
   RUNG wire#powerrail
      { S7_Templates := "SrcType := Int" } EQ_Contact(in1 := "INTERLOCK DB".BUFF."DPT-201", in2 := 2)
      { S7_Templates := "time_type := Time" } "IEC_Timer_0_DB_145".TOF(pt := T#2S, et =>)
      wire#w1
      Coil( "ALARM DB"."DPT-201 HIGH" )
   END_RUNG
   RUNG wire#w1
      P_Trig( "P_TRIG".ARR[73] )
      S_Coil( "OUTPUT MAPPING DB"."HOOTER RESET" )
   END_RUNG
   // the same network as SCL:
   "IEC_Timer_0_DB_145".TOF(IN := "INTERLOCK DB".BUFF."DPT-201" = 2, PT := T#2S);
   "ALARM DB"."DPT-201 HIGH" := "IEC_Timer_0_DB_145".Q;
   #_w1 := "IEC_Timer_0_DB_145".Q AND NOT "P_TRIG".ARR[73];   // rising edge
   "P_TRIG".ARR[73] := "IEC_Timer_0_DB_145".Q;
   IF #_w1 THEN "OUTPUT MAPPING DB"."HOOTER RESET" := TRUE; END_IF;
END_REGION

REGION Network 75: pHIT-601 LOW
   RUNG wire#powerrail
      { S7_Templates := "SrcType := Int" } EQ_Contact(in1 := "INTERLOCK DB".BUFF."pHIT-601 HIGH/LOW", in2 := 1)
      wire#w1
      Coil( "ALARM DB"."NRMB PRODUCT OUT pHIT-601 LOW" )
   END_RUNG
   RUNG wire#w1
      P_Trig( "P_TRIG".ARR[74] )
      S_Coil( "OUTPUT MAPPING DB"."HOOTER RESET" )
   END_RUNG
   // the same network as SCL:
   "ALARM DB"."NRMB PRODUCT OUT pHIT-601 LOW" := "INTERLOCK DB".BUFF."pHIT-601 HIGH/LOW" = 1;
   #_w1 := "ALARM DB"."NRMB PRODUCT OUT pHIT-601 LOW" AND NOT "P_TRIG".ARR[74];   // rising edge
   "P_TRIG".ARR[74] := "ALARM DB"."NRMB PRODUCT OUT pHIT-601 LOW";
   IF #_w1 THEN "OUTPUT MAPPING DB"."HOOTER RESET" := TRUE; END_IF;
END_REGION

REGION Network 76: pHIT-601HIGH
   RUNG wire#powerrail
      { S7_Templates := "SrcType := Int" } EQ_Contact(in1 := "INTERLOCK DB".BUFF."pHIT-601 HIGH/LOW", in2 := 2)
      wire#w1
      Coil( "ALARM DB"."NRMB PRODUCT OUT pHIT-601 HIGH" )
   END_RUNG
   RUNG wire#w1
      P_Trig( "P_TRIG".ARR[75] )
      S_Coil( "OUTPUT MAPPING DB"."HOOTER RESET" )
   END_RUNG
   // the same network as SCL:
   "ALARM DB"."NRMB PRODUCT OUT pHIT-601 HIGH" := "INTERLOCK DB".BUFF."pHIT-601 HIGH/LOW" = 2;
   #_w1 := "ALARM DB"."NRMB PRODUCT OUT pHIT-601 HIGH" AND NOT "P_TRIG".ARR[75];   // rising edge
   "P_TRIG".ARR[75] := "ALARM DB"."NRMB PRODUCT OUT pHIT-601 HIGH";
   IF #_w1 THEN "OUTPUT MAPPING DB"."HOOTER RESET" := TRUE; END_IF;
END_REGION

REGION Network 77: RIT-601 HIGH
   RUNG wire#powerrail
      { S7_Templates := "SrcType := Int" } EQ_Contact(in1 := "INTERLOCK DB".BUFF."RIT-601 HIGH BUFF", in2 := 2)
      wire#w1
      Coil( "ALARM DB"."NRMB PRODUCT OUT RIT-601 HIGH" )
   END_RUNG
   RUNG wire#w1
      P_Trig( "P_TRIG".ARR[76] )
      S_Coil( "OUTPUT MAPPING DB"."HOOTER RESET" )
   END_RUNG
   // the same network as SCL:
   "ALARM DB"."NRMB PRODUCT OUT RIT-601 HIGH" := "INTERLOCK DB".BUFF."RIT-601 HIGH BUFF" = 2;
   #_w1 := "ALARM DB"."NRMB PRODUCT OUT RIT-601 HIGH" AND NOT "P_TRIG".ARR[76];   // rising edge
   "P_TRIG".ARR[76] := "ALARM DB"."NRMB PRODUCT OUT RIT-601 HIGH";
   IF #_w1 THEN "OUTPUT MAPPING DB"."HOOTER RESET" := TRUE; END_IF;
END_REGION

REGION Network 78: RIT-601 HIGH HIGH
   RUNG wire#powerrail
      Contact( "TIMING_MIN_DB_6".DONE )
      { S7_Templates := "time_type := Time" } "IEC_Timer_0_DB_137".TOF(pt := T#2S, et =>)
      wire#w1
      Coil( "ALARM DB"."RIT-601 HIGH_SET VALIDATION TIME OVER_(SYSTEM STOP)" )
   END_RUNG
   RUNG wire#w1
      P_Trig( "P_TRIG".ARR[77] )
      S_Coil( "OUTPUT MAPPING DB"."HOOTER RESET" )
   END_RUNG
   // the same network as SCL:
   "IEC_Timer_0_DB_137".TOF(IN := "TIMING_MIN_DB_6".DONE, PT := T#2S);
   "ALARM DB"."RIT-601 HIGH_SET VALIDATION TIME OVER_(SYSTEM STOP)" := "IEC_Timer_0_DB_137".Q;
   #_w1 := "IEC_Timer_0_DB_137".Q AND NOT "P_TRIG".ARR[77];   // rising edge
   "P_TRIG".ARR[77] := "IEC_Timer_0_DB_137".Q;
   IF #_w1 THEN "OUTPUT MAPPING DB"."HOOTER RESET" := TRUE; END_IF;
END_REGION

REGION Network 79
   RUNG wire#powerrail
      Contact( "INTERLOCK DB".BUFF."UV ONLY ALARM" )
      wire#w1
      Coil( "ALARM DB"."UV-601 INTENSITY LOW" )
   END_RUNG
   RUNG wire#w1
      P_Trig( "P_TRIG".ARR[78] )
      S_Coil( "OUTPUT MAPPING DB"."HOOTER RESET" )
   END_RUNG
   // the same network as SCL:
   "ALARM DB"."UV-601 INTENSITY LOW" := "INTERLOCK DB".BUFF."UV ONLY ALARM";
   #_w1 := "INTERLOCK DB".BUFF."UV ONLY ALARM" AND NOT "P_TRIG".ARR[78];   // rising edge
   "P_TRIG".ARR[78] := "INTERLOCK DB".BUFF."UV ONLY ALARM";
   IF #_w1 THEN "OUTPUT MAPPING DB"."HOOTER RESET" := TRUE; END_IF;
END_REGION
END_FUNCTION

FUNCTION "DATE&TIMES" : Void   // FC9, LAD
{ S7_Optimized_Access := 'TRUE' }
// stored: SetENOAutomatically false
BEGIN

REGION Network 1
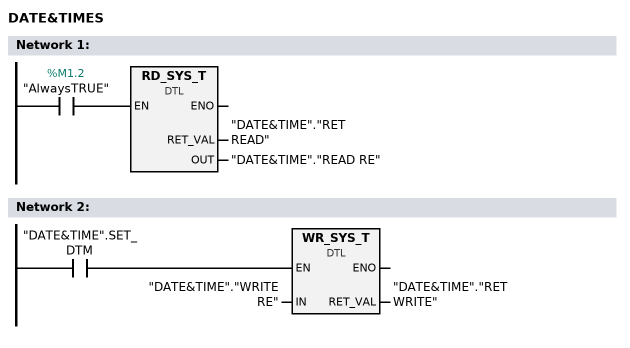
   RUNG wire#powerrail
      Contact( "AlwaysTRUE" )
      { S7_Templates := "date_type := DTL" } RD_SYS_T(RET_VAL => "DATE&TIME"."RET READ", OUT => "DATE&TIME"."READ RE")
   END_RUNG
   // the same network as SCL:
   IF "AlwaysTRUE" THEN "DATE&TIME"."RET READ" := RD_SYS_T(OUT => "DATE&TIME"."READ RE"); END_IF;
END_REGION

REGION Network 2
   RUNG wire#powerrail
      Contact( "DATE&TIME".SET_DTM )
      { S7_Templates := "date_type := DTL" } WR_SYS_T(IN := "DATE&TIME"."WRITE RE", RET_VAL => "DATE&TIME"."RET WRITE")
   END_RUNG
   // the same network as SCL:
   IF "DATE&TIME".SET_DTM THEN "DATE&TIME"."RET WRITE" := WR_SYS_T(IN := "DATE&TIME"."WRITE RE"); END_IF;
END_REGION
END_FUNCTION

FUNCTION "AI SCALING" : Void   // FC5, LAD
{ S7_Optimized_Access := 'TRUE' }
// stored: SetENOAutomatically false
   VAR_TEMP   // added for the SCL form of the ladder/FBD networks
      _w1 : Bool;
   END_VAR
BEGIN

REGION Network 1: LEVEL TRANSMITTER-101 ANALOG
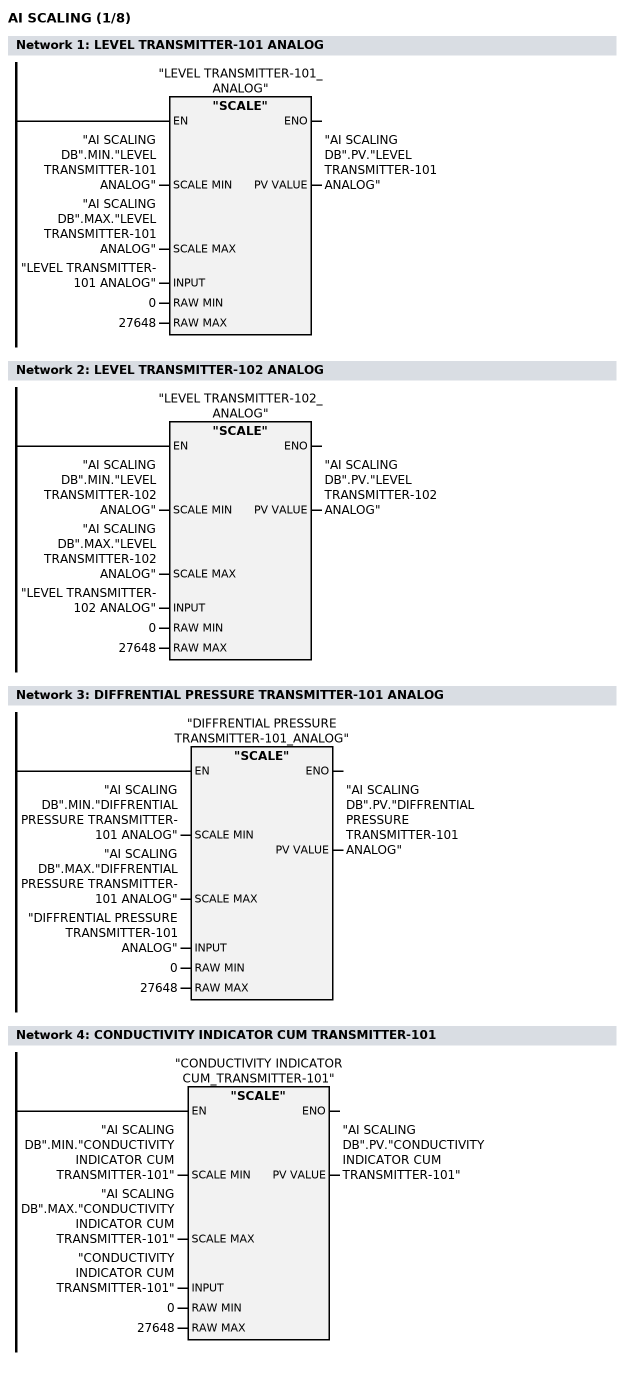
   RUNG wire#powerrail
      "LEVEL TRANSMITTER-101_ANALOG"("SCALE MIN" := "AI SCALING DB".MIN."LEVEL TRANSMITTER-101 ANALOG", "SCALE MAX" := "AI SCALING DB".MAX."LEVEL TRANSMITTER-101 ANALOG", INPUT := "LEVEL TRANSMITTER-101 ANALOG", "RAW MIN" := 0, "RAW MAX" := 27648, "PV VALUE" => "AI SCALING DB".PV."LEVEL TRANSMITTER-101 ANALOG")
   END_RUNG
   // the same network as SCL:
   "LEVEL TRANSMITTER-101_ANALOG"("SCALE MIN" := "AI SCALING DB".MIN."LEVEL TRANSMITTER-101 ANALOG",   // "SCALE"
                           "SCALE MAX" := "AI SCALING DB".MAX."LEVEL TRANSMITTER-101 ANALOG",
                           INPUT := "LEVEL TRANSMITTER-101 ANALOG",
                           "RAW MIN" := 0,
                           "RAW MAX" := 27648,
                           "PV VALUE" => "AI SCALING DB".PV."LEVEL TRANSMITTER-101 ANALOG");
END_REGION

REGION Network 2: LEVEL TRANSMITTER-102 ANALOG
   RUNG wire#powerrail
      "LEVEL TRANSMITTER-102_ANALOG"("SCALE MIN" := "AI SCALING DB".MIN."LEVEL TRANSMITTER-102 ANALOG", "SCALE MAX" := "AI SCALING DB".MAX."LEVEL TRANSMITTER-102 ANALOG", INPUT := "LEVEL TRANSMITTER-102 ANALOG", "RAW MIN" := 0, "RAW MAX" := 27648, "PV VALUE" => "AI SCALING DB".PV."LEVEL TRANSMITTER-102 ANALOG")
   END_RUNG
   // the same network as SCL:
   "LEVEL TRANSMITTER-102_ANALOG"("SCALE MIN" := "AI SCALING DB".MIN."LEVEL TRANSMITTER-102 ANALOG",   // "SCALE"
                           "SCALE MAX" := "AI SCALING DB".MAX."LEVEL TRANSMITTER-102 ANALOG",
                           INPUT := "LEVEL TRANSMITTER-102 ANALOG",
                           "RAW MIN" := 0,
                           "RAW MAX" := 27648,
                           "PV VALUE" => "AI SCALING DB".PV."LEVEL TRANSMITTER-102 ANALOG");
END_REGION

REGION Network 3: DIFFRENTIAL PRESSURE TRANSMITTER-101 ANALOG
   RUNG wire#powerrail
      "DIFFRENTIAL PRESSURE TRANSMITTER-101_ANALOG"("SCALE MIN" := "AI SCALING DB".MIN."DIFFRENTIAL PRESSURE TRANSMITTER-101 ANALOG", "SCALE MAX" := "AI SCALING DB".MAX."DIFFRENTIAL PRESSURE TRANSMITTER-101 ANALOG", INPUT := "DIFFRENTIAL PRESSURE TRANSMITTER-101 ANALOG", "RAW MIN" := 0, "RAW MAX" := 27648, "PV VALUE" => "AI SCALING DB".PV."DIFFRENTIAL PRESSURE TRANSMITTER-101 ANALOG")
   END_RUNG
   // the same network as SCL:
   "DIFFRENTIAL PRESSURE TRANSMITTER-101_ANALOG"("SCALE MIN" := "AI SCALING DB".MIN."DIFFRENTIAL PRESSURE TRANSMITTER-101 ANALOG",   // "SCALE"
                           "SCALE MAX" := "AI SCALING DB".MAX."DIFFRENTIAL PRESSURE TRANSMITTER-101 ANALOG",
                           INPUT := "DIFFRENTIAL PRESSURE TRANSMITTER-101 ANALOG",
                           "RAW MIN" := 0,
                           "RAW MAX" := 27648,
                           "PV VALUE" => "AI SCALING DB".PV."DIFFRENTIAL PRESSURE TRANSMITTER-101 ANALOG");
END_REGION

REGION Network 4: CONDUCTIVITY INDICATOR CUM TRANSMITTER-101
   RUNG wire#powerrail
      "CONDUCTIVITY INDICATOR CUM_TRANSMITTER-101"("SCALE MIN" := "AI SCALING DB".MIN."CONDUCTIVITY INDICATOR CUM TRANSMITTER-101", "SCALE MAX" := "AI SCALING DB".MAX."CONDUCTIVITY INDICATOR CUM TRANSMITTER-101", INPUT := "CONDUCTIVITY INDICATOR CUM TRANSMITTER-101", "RAW MIN" := 0, "RAW MAX" := 27648, "PV VALUE" => "AI SCALING DB".PV."CONDUCTIVITY INDICATOR CUM TRANSMITTER-101")
   END_RUNG
   // the same network as SCL:
   "CONDUCTIVITY INDICATOR CUM_TRANSMITTER-101"("SCALE MIN" := "AI SCALING DB".MIN."CONDUCTIVITY INDICATOR CUM TRANSMITTER-101",   // "SCALE"
                           "SCALE MAX" := "AI SCALING DB".MAX."CONDUCTIVITY INDICATOR CUM TRANSMITTER-101",
                           INPUT := "CONDUCTIVITY INDICATOR CUM TRANSMITTER-101",
                           "RAW MIN" := 0,
                           "RAW MAX" := 27648,
                           "PV VALUE" => "AI SCALING DB".PV."CONDUCTIVITY INDICATOR CUM TRANSMITTER-101");
END_REGION

REGION Network 5: DIFFRENTIAL PRESSURE TRANSMITTER-201
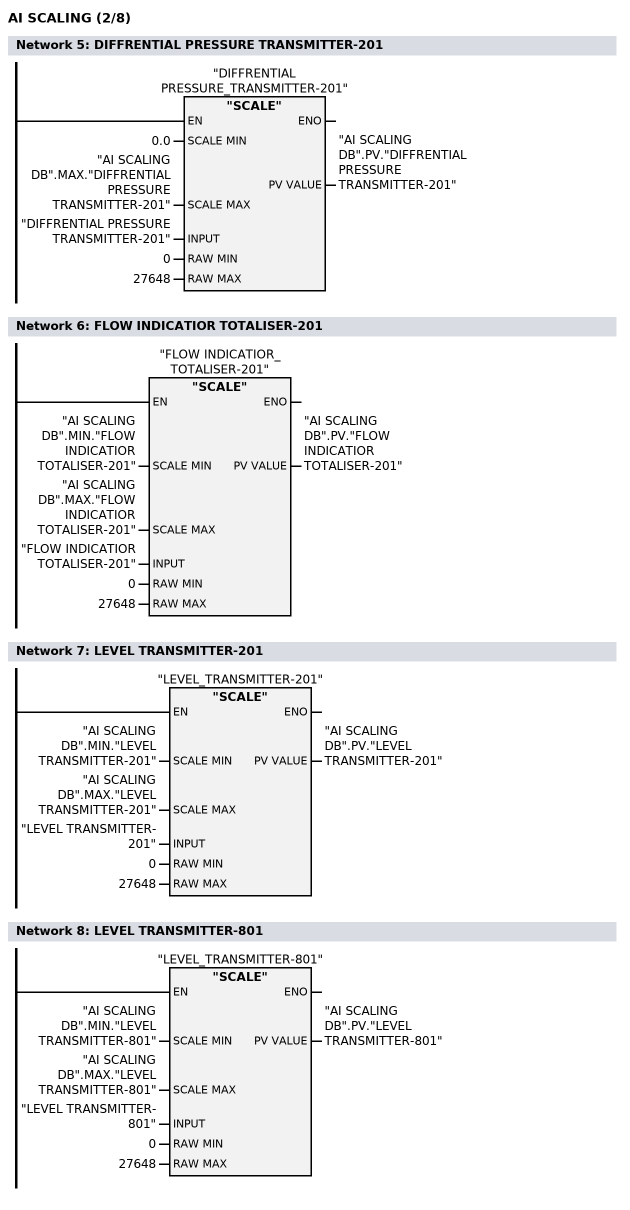
   RUNG wire#powerrail
      "DIFFRENTIAL PRESSURE_TRANSMITTER-201"("SCALE MIN" := 0.0, "SCALE MAX" := "AI SCALING DB".MAX."DIFFRENTIAL PRESSURE TRANSMITTER-201", INPUT := "DIFFRENTIAL PRESSURE TRANSMITTER-201", "RAW MIN" := 0, "RAW MAX" := 27648, "PV VALUE" => "AI SCALING DB".PV."DIFFRENTIAL PRESSURE TRANSMITTER-201")
   END_RUNG
   // the same network as SCL:
   "DIFFRENTIAL PRESSURE_TRANSMITTER-201"("SCALE MIN" := 0.0,   // "SCALE"
                           "SCALE MAX" := "AI SCALING DB".MAX."DIFFRENTIAL PRESSURE TRANSMITTER-201",
                           INPUT := "DIFFRENTIAL PRESSURE TRANSMITTER-201",
                           "RAW MIN" := 0,
                           "RAW MAX" := 27648,
                           "PV VALUE" => "AI SCALING DB".PV."DIFFRENTIAL PRESSURE TRANSMITTER-201");
END_REGION

REGION Network 6: FLOW INDICATIOR TOTALISER-201
   RUNG wire#powerrail
      "FLOW INDICATIOR_TOTALISER-201"("SCALE MIN" := "AI SCALING DB".MIN."FLOW INDICATIOR TOTALISER-201", "SCALE MAX" := "AI SCALING DB".MAX."FLOW INDICATIOR TOTALISER-201", INPUT := "FLOW INDICATIOR TOTALISER-201", "RAW MIN" := 0, "RAW MAX" := 27648, "PV VALUE" => "AI SCALING DB".PV."FLOW INDICATIOR TOTALISER-201")
   END_RUNG
   // the same network as SCL:
   "FLOW INDICATIOR_TOTALISER-201"("SCALE MIN" := "AI SCALING DB".MIN."FLOW INDICATIOR TOTALISER-201",   // "SCALE"
                           "SCALE MAX" := "AI SCALING DB".MAX."FLOW INDICATIOR TOTALISER-201",
                           INPUT := "FLOW INDICATIOR TOTALISER-201",
                           "RAW MIN" := 0,
                           "RAW MAX" := 27648,
                           "PV VALUE" => "AI SCALING DB".PV."FLOW INDICATIOR TOTALISER-201");
END_REGION

REGION Network 7: LEVEL TRANSMITTER-201
   RUNG wire#powerrail
      "LEVEL_TRANSMITTER-201"("SCALE MIN" := "AI SCALING DB".MIN."LEVEL TRANSMITTER-201", "SCALE MAX" := "AI SCALING DB".MAX."LEVEL TRANSMITTER-201", INPUT := "LEVEL TRANSMITTER-201", "RAW MIN" := 0, "RAW MAX" := 27648, "PV VALUE" => "AI SCALING DB".PV."LEVEL TRANSMITTER-201")
   END_RUNG
   // the same network as SCL:
   "LEVEL_TRANSMITTER-201"("SCALE MIN" := "AI SCALING DB".MIN."LEVEL TRANSMITTER-201",   // "SCALE"
                           "SCALE MAX" := "AI SCALING DB".MAX."LEVEL TRANSMITTER-201",
                           INPUT := "LEVEL TRANSMITTER-201",
                           "RAW MIN" := 0,
                           "RAW MAX" := 27648,
                           "PV VALUE" => "AI SCALING DB".PV."LEVEL TRANSMITTER-201");
END_REGION

REGION Network 8: LEVEL TRANSMITTER-801
   RUNG wire#powerrail
      "LEVEL_TRANSMITTER-801"("SCALE MIN" := "AI SCALING DB".MIN."LEVEL TRANSMITTER-801", "SCALE MAX" := "AI SCALING DB".MAX."LEVEL TRANSMITTER-801", INPUT := "LEVEL TRANSMITTER-801", "RAW MIN" := 0, "RAW MAX" := 27648, "PV VALUE" => "AI SCALING DB".PV."LEVEL TRANSMITTER-801")
   END_RUNG
   // the same network as SCL:
   "LEVEL_TRANSMITTER-801"("SCALE MIN" := "AI SCALING DB".MIN."LEVEL TRANSMITTER-801",   // "SCALE"
                           "SCALE MAX" := "AI SCALING DB".MAX."LEVEL TRANSMITTER-801",
                           INPUT := "LEVEL TRANSMITTER-801",
                           "RAW MIN" := 0,
                           "RAW MAX" := 27648,
                           "PV VALUE" => "AI SCALING DB".PV."LEVEL TRANSMITTER-801");
END_REGION

REGION Network 9: RESISTIVITY CUM TRANSMITTER 601
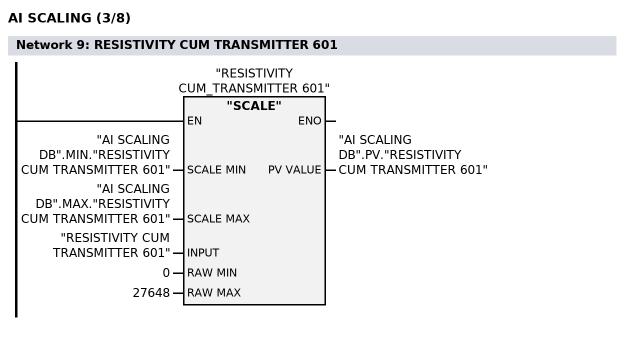
   RUNG wire#powerrail
      "RESISTIVITY CUM_TRANSMITTER 601"("SCALE MIN" := "AI SCALING DB".MIN."RESISTIVITY CUM TRANSMITTER 601", "SCALE MAX" := "AI SCALING DB".MAX."RESISTIVITY CUM TRANSMITTER 601", INPUT := "RESISTIVITY CUM TRANSMITTER 601", "RAW MIN" := 0, "RAW MAX" := 27648, "PV VALUE" => "AI SCALING DB".PV."RESISTIVITY CUM TRANSMITTER 601")
   END_RUNG
   // the same network as SCL:
   "RESISTIVITY CUM_TRANSMITTER 601"("SCALE MIN" := "AI SCALING DB".MIN."RESISTIVITY CUM TRANSMITTER 601",   // "SCALE"
                           "SCALE MAX" := "AI SCALING DB".MAX."RESISTIVITY CUM TRANSMITTER 601",
                           INPUT := "RESISTIVITY CUM TRANSMITTER 601",
                           "RAW MIN" := 0,
                           "RAW MAX" := 27648,
                           "PV VALUE" => "AI SCALING DB".PV."RESISTIVITY CUM TRANSMITTER 601");
END_REGION

REGION Network 10: PRESSURE TRANSMITTER 601
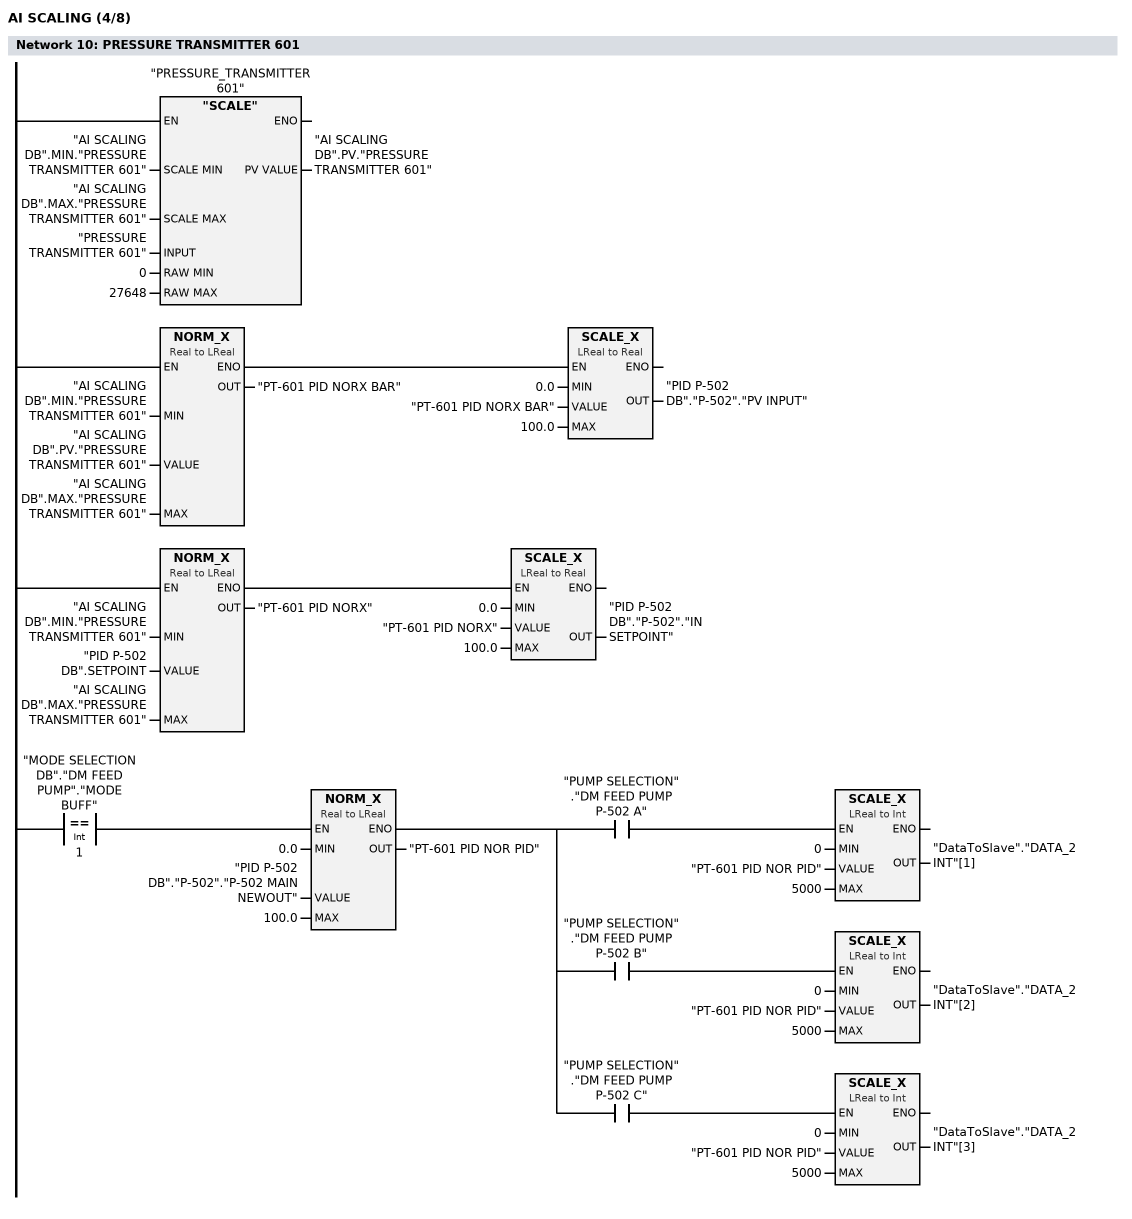
   RUNG wire#powerrail
      "PRESSURE_TRANSMITTER 601"("SCALE MIN" := "AI SCALING DB".MIN."PRESSURE TRANSMITTER 601", "SCALE MAX" := "AI SCALING DB".MAX."PRESSURE TRANSMITTER 601", INPUT := "PRESSURE TRANSMITTER 601", "RAW MIN" := 0, "RAW MAX" := 27648, "PV VALUE" => "AI SCALING DB".PV."PRESSURE TRANSMITTER 601")
   END_RUNG
   RUNG wire#powerrail
      { S7_Templates := "[SrcType := Real, DestType := LReal]" } Normalize(min := "AI SCALING DB".MIN."PRESSURE TRANSMITTER 601", value := "AI SCALING DB".PV."PRESSURE TRANSMITTER 601", max := "AI SCALING DB".MAX."PRESSURE TRANSMITTER 601", out => "PT-601 PID NORX BAR")
      { S7_Templates := "[SrcType := LReal, DestType := Real]" } Scale(min := 0.0, value := "PT-601 PID NORX BAR", max := 100.0, out => "PID P-502 DB"."P-502"."PV INPUT")
   END_RUNG
   RUNG wire#powerrail
      { S7_Templates := "[SrcType := Real, DestType := LReal]" } Normalize(min := "AI SCALING DB".MIN."PRESSURE TRANSMITTER 601", value := "PID P-502 DB".SETPOINT, max := "AI SCALING DB".MAX."PRESSURE TRANSMITTER 601", out => "PT-601 PID NORX")
      { S7_Templates := "[SrcType := LReal, DestType := Real]" } Scale(min := 0.0, value := "PT-601 PID NORX", max := 100.0, out => "PID P-502 DB"."P-502"."IN SETPOINT")
   END_RUNG
   RUNG wire#powerrail
      { S7_Templates := "SrcType := Int" } EQ_Contact(in1 := "MODE SELECTION DB"."DM FEED PUMP"."MODE BUFF", in2 := 1)
      { S7_Templates := "[SrcType := Real, DestType := LReal]" } Normalize(min := 0.0, value := "PID P-502 DB"."P-502"."P-502 MAIN NEWOUT", max := 100.0, out => "PT-601 PID NOR PID")
      wire#w1
      Contact( "PUMP SELECTION"."DM FEED PUMP P-502 A" )
      { S7_Templates := "[SrcType := LReal, DestType := Int]" } Scale(min := 0, value := "PT-601 PID NOR PID", max := 5000, out => "DataToSlave"."DATA_2 INT"[1])
   END_RUNG
   RUNG wire#w1
      Contact( "PUMP SELECTION"."DM FEED PUMP P-502 B" )
      { S7_Templates := "[SrcType := LReal, DestType := Int]" } Scale(min := 0, value := "PT-601 PID NOR PID", max := 5000, out => "DataToSlave"."DATA_2 INT"[2])
   END_RUNG
   RUNG wire#w1
      Contact( "PUMP SELECTION"."DM FEED PUMP P-502 C" )
      { S7_Templates := "[SrcType := LReal, DestType := Int]" } Scale(min := 0, value := "PT-601 PID NOR PID", max := 5000, out => "DataToSlave"."DATA_2 INT"[3])
   END_RUNG
   // the same network as SCL:
   "PRESSURE_TRANSMITTER 601"("SCALE MIN" := "AI SCALING DB".MIN."PRESSURE TRANSMITTER 601",   // "SCALE"
                           "SCALE MAX" := "AI SCALING DB".MAX."PRESSURE TRANSMITTER 601",
                           INPUT := "PRESSURE TRANSMITTER 601",
                           "RAW MIN" := 0,
                           "RAW MAX" := 27648,
                           "PV VALUE" => "AI SCALING DB".PV."PRESSURE TRANSMITTER 601");
   "PT-601 PID NORX BAR" := NORM_X(MIN := "AI SCALING DB".MIN."PRESSURE TRANSMITTER 601", VALUE := "AI SCALING DB".PV."PRESSURE TRANSMITTER 601", MAX := "AI SCALING DB".MAX."PRESSURE TRANSMITTER 601");
   "PID P-502 DB"."P-502"."PV INPUT" := SCALE_X(MIN := 0.0, VALUE := "PT-601 PID NORX BAR", MAX := 100.0);
   "PT-601 PID NORX" := NORM_X(MIN := "AI SCALING DB".MIN."PRESSURE TRANSMITTER 601", VALUE := "PID P-502 DB".SETPOINT, MAX := "AI SCALING DB".MAX."PRESSURE TRANSMITTER 601");
   "PID P-502 DB"."P-502"."IN SETPOINT" := SCALE_X(MIN := 0.0, VALUE := "PT-601 PID NORX", MAX := 100.0);
   #_w1 := "MODE SELECTION DB"."DM FEED PUMP"."MODE BUFF" = 1;
   IF #_w1 THEN
       "PT-601 PID NOR PID" := NORM_X(MIN := 0.0, VALUE := "PID P-502 DB"."P-502"."P-502 MAIN NEWOUT", MAX := 100.0);
   END_IF;
   IF #_w1 AND "PUMP SELECTION"."DM FEED PUMP P-502 A" THEN
       "DataToSlave"."DATA_2 INT"[1] := SCALE_X(MIN := 0, VALUE := "PT-601 PID NOR PID", MAX := 5000);
   END_IF;
   IF #_w1 AND "PUMP SELECTION"."DM FEED PUMP P-502 B" THEN
       "DataToSlave"."DATA_2 INT"[2] := SCALE_X(MIN := 0, VALUE := "PT-601 PID NOR PID", MAX := 5000);
   END_IF;
   IF #_w1 AND "PUMP SELECTION"."DM FEED PUMP P-502 C" THEN
       "DataToSlave"."DATA_2 INT"[3] := SCALE_X(MIN := 0, VALUE := "PT-601 PID NOR PID", MAX := 5000);
   END_IF;
END_REGION

REGION Network 11: FLOW INDICATIOR TOTALISER 601
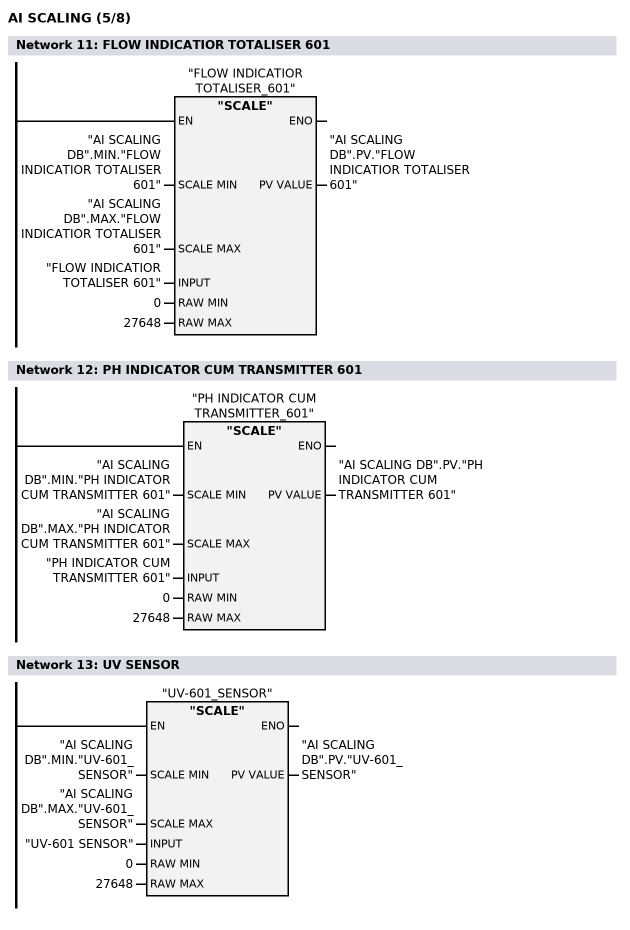
   RUNG wire#powerrail
      "FLOW INDICATIOR TOTALISER_601"("SCALE MIN" := "AI SCALING DB".MIN."FLOW INDICATIOR TOTALISER 601", "SCALE MAX" := "AI SCALING DB".MAX."FLOW INDICATIOR TOTALISER 601", INPUT := "FLOW INDICATIOR TOTALISER 601", "RAW MIN" := 0, "RAW MAX" := 27648, "PV VALUE" => "AI SCALING DB".PV."FLOW INDICATIOR TOTALISER 601")
   END_RUNG
   // the same network as SCL:
   "FLOW INDICATIOR TOTALISER_601"("SCALE MIN" := "AI SCALING DB".MIN."FLOW INDICATIOR TOTALISER 601",   // "SCALE"
                           "SCALE MAX" := "AI SCALING DB".MAX."FLOW INDICATIOR TOTALISER 601",
                           INPUT := "FLOW INDICATIOR TOTALISER 601",
                           "RAW MIN" := 0,
                           "RAW MAX" := 27648,
                           "PV VALUE" => "AI SCALING DB".PV."FLOW INDICATIOR TOTALISER 601");
END_REGION

REGION Network 12: PH INDICATOR CUM TRANSMITTER 601
   RUNG wire#powerrail
      "PH INDICATOR CUM TRANSMITTER_601"("SCALE MIN" := "AI SCALING DB".MIN."PH INDICATOR CUM TRANSMITTER 601", "SCALE MAX" := "AI SCALING DB".MAX."PH INDICATOR CUM TRANSMITTER 601", INPUT := "PH INDICATOR CUM TRANSMITTER 601", "RAW MIN" := 0, "RAW MAX" := 27648, "PV VALUE" => "AI SCALING DB".PV."PH INDICATOR CUM TRANSMITTER 601")
   END_RUNG
   // the same network as SCL:
   "PH INDICATOR CUM TRANSMITTER_601"("SCALE MIN" := "AI SCALING DB".MIN."PH INDICATOR CUM TRANSMITTER 601",   // "SCALE"
                           "SCALE MAX" := "AI SCALING DB".MAX."PH INDICATOR CUM TRANSMITTER 601",
                           INPUT := "PH INDICATOR CUM TRANSMITTER 601",
                           "RAW MIN" := 0,
                           "RAW MAX" := 27648,
                           "PV VALUE" => "AI SCALING DB".PV."PH INDICATOR CUM TRANSMITTER 601");
END_REGION

REGION Network 13: UV SENSOR
   RUNG wire#powerrail
      "UV-601_SENSOR"("SCALE MIN" := "AI SCALING DB".MIN."UV-601_SENSOR", "SCALE MAX" := "AI SCALING DB".MAX."UV-601_SENSOR", INPUT := "UV-601 SENSOR", "RAW MIN" := 0, "RAW MAX" := 27648, "PV VALUE" => "AI SCALING DB".PV."UV-601_SENSOR")
   END_RUNG
   // the same network as SCL:
   "UV-601_SENSOR"("SCALE MIN" := "AI SCALING DB".MIN."UV-601_SENSOR",   // "SCALE"
                   "SCALE MAX" := "AI SCALING DB".MAX."UV-601_SENSOR",
                   INPUT := "UV-601 SENSOR",
                   "RAW MIN" := 0,
                   "RAW MAX" := 27648,
                   "PV VALUE" => "AI SCALING DB".PV."UV-601_SENSOR");
END_REGION

REGION Network 16: LT-101 BUFFER
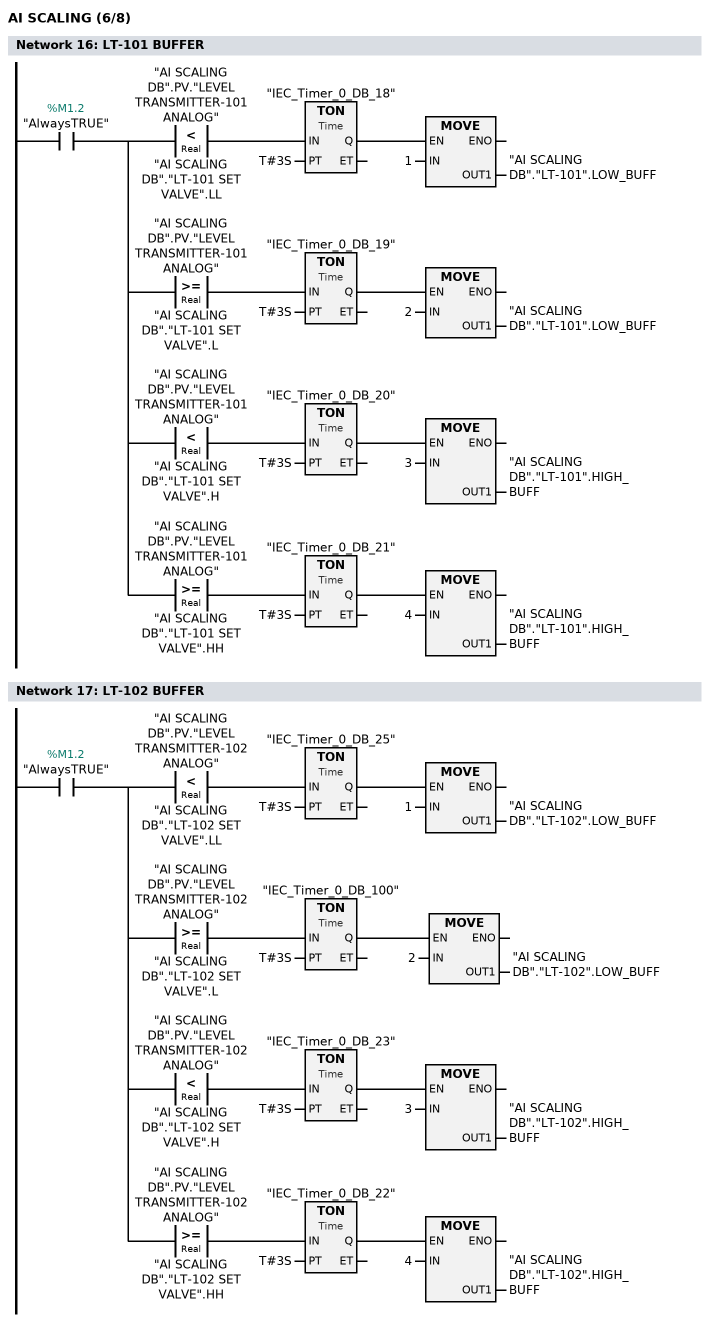
   RUNG wire#powerrail
      Contact( "AlwaysTRUE" )
      wire#w1
      { S7_Templates := "SrcType := Real" } LT_Contact(in1 := "AI SCALING DB".PV."LEVEL TRANSMITTER-101 ANALOG", in2 := "AI SCALING DB"."LT-101 SET VALVE".LL)
      { S7_Templates := "time_type := Time" } "IEC_Timer_0_DB_18".TON(pt := T#3S, et =>)
      Move(in := 1, out1 => "AI SCALING DB"."LT-101".LOW_BUFF)
   END_RUNG
   RUNG wire#w1
      { S7_Templates := "SrcType := Real" } GE_Contact(in1 := "AI SCALING DB".PV."LEVEL TRANSMITTER-101 ANALOG", in2 := "AI SCALING DB"."LT-101 SET VALVE".L)
      { S7_Templates := "time_type := Time" } "IEC_Timer_0_DB_19".TON(pt := T#3S, et =>)
      Move(in := 2, out1 => "AI SCALING DB"."LT-101".LOW_BUFF)
   END_RUNG
   RUNG wire#w1
      { S7_Templates := "SrcType := Real" } LT_Contact(in1 := "AI SCALING DB".PV."LEVEL TRANSMITTER-101 ANALOG", in2 := "AI SCALING DB"."LT-101 SET VALVE".H)
      { S7_Templates := "time_type := Time" } "IEC_Timer_0_DB_20".TON(pt := T#3S, et =>)
      Move(in := 3, out1 => "AI SCALING DB"."LT-101".HIGH_BUFF)
   END_RUNG
   RUNG wire#w1
      { S7_Templates := "SrcType := Real" } GE_Contact(in1 := "AI SCALING DB".PV."LEVEL TRANSMITTER-101 ANALOG", in2 := "AI SCALING DB"."LT-101 SET VALVE".HH)
      { S7_Templates := "time_type := Time" } "IEC_Timer_0_DB_21".TON(pt := T#3S, et =>)
      Move(in := 4, out1 => "AI SCALING DB"."LT-101".HIGH_BUFF)
   END_RUNG
   // the same network as SCL:
   "IEC_Timer_0_DB_18".TON(IN := "AlwaysTRUE" AND ("AI SCALING DB".PV."LEVEL TRANSMITTER-101 ANALOG" < "AI SCALING DB"."LT-101 SET VALVE".LL),
                           PT := T#3S);
   IF "IEC_Timer_0_DB_18".Q THEN "AI SCALING DB"."LT-101".LOW_BUFF := 1; END_IF;
   "IEC_Timer_0_DB_19".TON(IN := "AlwaysTRUE" AND ("AI SCALING DB".PV."LEVEL TRANSMITTER-101 ANALOG" >= "AI SCALING DB"."LT-101 SET VALVE".L),
                           PT := T#3S);
   IF "IEC_Timer_0_DB_19".Q THEN "AI SCALING DB"."LT-101".LOW_BUFF := 2; END_IF;
   "IEC_Timer_0_DB_20".TON(IN := "AlwaysTRUE" AND ("AI SCALING DB".PV."LEVEL TRANSMITTER-101 ANALOG" < "AI SCALING DB"."LT-101 SET VALVE".H),
                           PT := T#3S);
   IF "IEC_Timer_0_DB_20".Q THEN "AI SCALING DB"."LT-101".HIGH_BUFF := 3; END_IF;
   "IEC_Timer_0_DB_21".TON(IN := "AlwaysTRUE" AND ("AI SCALING DB".PV."LEVEL TRANSMITTER-101 ANALOG" >= "AI SCALING DB"."LT-101 SET VALVE".HH),
                           PT := T#3S);
   IF "IEC_Timer_0_DB_21".Q THEN "AI SCALING DB"."LT-101".HIGH_BUFF := 4; END_IF;
END_REGION

REGION Network 17: LT-102 BUFFER
   RUNG wire#powerrail
      Contact( "AlwaysTRUE" )
      wire#w1
      { S7_Templates := "SrcType := Real" } LT_Contact(in1 := "AI SCALING DB".PV."LEVEL TRANSMITTER-102 ANALOG", in2 := "AI SCALING DB"."LT-102 SET VALVE".LL)
      { S7_Templates := "time_type := Time" } "IEC_Timer_0_DB_25".TON(pt := T#3S, et =>)
      Move(in := 1, out1 => "AI SCALING DB"."LT-102".LOW_BUFF)
   END_RUNG
   RUNG wire#w1
      { S7_Templates := "SrcType := Real" } GE_Contact(in1 := "AI SCALING DB".PV."LEVEL TRANSMITTER-102 ANALOG", in2 := "AI SCALING DB"."LT-102 SET VALVE".L)
      { S7_Templates := "time_type := Time" } "IEC_Timer_0_DB_100".TON(pt := T#3S, et =>)
      Move(in := 2, out1 => "AI SCALING DB"."LT-102".LOW_BUFF)
   END_RUNG
   RUNG wire#w1
      { S7_Templates := "SrcType := Real" } LT_Contact(in1 := "AI SCALING DB".PV."LEVEL TRANSMITTER-102 ANALOG", in2 := "AI SCALING DB"."LT-102 SET VALVE".H)
      { S7_Templates := "time_type := Time" } "IEC_Timer_0_DB_23".TON(pt := T#3S, et =>)
      Move(in := 3, out1 => "AI SCALING DB"."LT-102".HIGH_BUFF)
   END_RUNG
   RUNG wire#w1
      { S7_Templates := "SrcType := Real" } GE_Contact(in1 := "AI SCALING DB".PV."LEVEL TRANSMITTER-102 ANALOG", in2 := "AI SCALING DB"."LT-102 SET VALVE".HH)
      { S7_Templates := "time_type := Time" } "IEC_Timer_0_DB_22".TON(pt := T#3S, et =>)
      Move(in := 4, out1 => "AI SCALING DB"."LT-102".HIGH_BUFF)
   END_RUNG
   // the same network as SCL:
   "IEC_Timer_0_DB_25".TON(IN := "AlwaysTRUE" AND ("AI SCALING DB".PV."LEVEL TRANSMITTER-102 ANALOG" < "AI SCALING DB"."LT-102 SET VALVE".LL),
                           PT := T#3S);
   IF "IEC_Timer_0_DB_25".Q THEN "AI SCALING DB"."LT-102".LOW_BUFF := 1; END_IF;
   "IEC_Timer_0_DB_100".TON(IN := "AlwaysTRUE" AND ("AI SCALING DB".PV."LEVEL TRANSMITTER-102 ANALOG" >= "AI SCALING DB"."LT-102 SET VALVE".L),
                           PT := T#3S);
   IF "IEC_Timer_0_DB_100".Q THEN "AI SCALING DB"."LT-102".LOW_BUFF := 2; END_IF;
   "IEC_Timer_0_DB_23".TON(IN := "AlwaysTRUE" AND ("AI SCALING DB".PV."LEVEL TRANSMITTER-102 ANALOG" < "AI SCALING DB"."LT-102 SET VALVE".H),
                           PT := T#3S);
   IF "IEC_Timer_0_DB_23".Q THEN "AI SCALING DB"."LT-102".HIGH_BUFF := 3; END_IF;
   "IEC_Timer_0_DB_22".TON(IN := "AlwaysTRUE" AND ("AI SCALING DB".PV."LEVEL TRANSMITTER-102 ANALOG" >= "AI SCALING DB"."LT-102 SET VALVE".HH),
                           PT := T#3S);
   IF "IEC_Timer_0_DB_22".Q THEN "AI SCALING DB"."LT-102".HIGH_BUFF := 4; END_IF;
END_REGION

REGION Network 18: LT-201 BUFFER
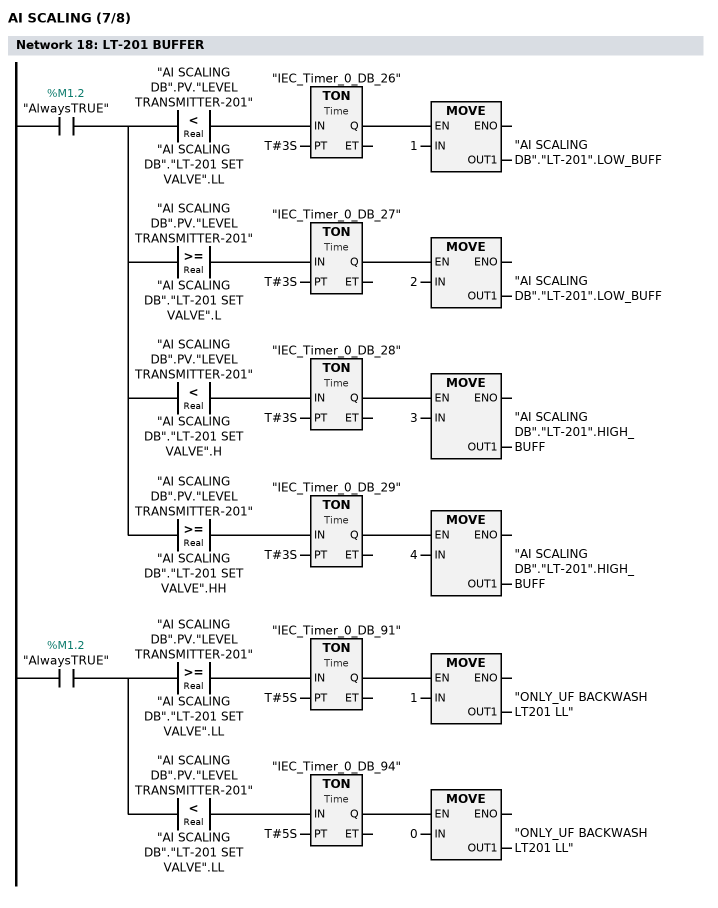
   RUNG wire#powerrail
      Contact( "AlwaysTRUE" )
      wire#w1
      { S7_Templates := "SrcType := Real" } LT_Contact(in1 := "AI SCALING DB".PV."LEVEL TRANSMITTER-201", in2 := "AI SCALING DB"."LT-201 SET VALVE".LL)
      { S7_Templates := "time_type := Time" } "IEC_Timer_0_DB_26".TON(pt := T#3S, et =>)
      Move(in := 1, out1 => "AI SCALING DB"."LT-201".LOW_BUFF)
   END_RUNG
   RUNG wire#w1
      { S7_Templates := "SrcType := Real" } GE_Contact(in1 := "AI SCALING DB".PV."LEVEL TRANSMITTER-201", in2 := "AI SCALING DB"."LT-201 SET VALVE".L)
      { S7_Templates := "time_type := Time" } "IEC_Timer_0_DB_27".TON(pt := T#3S, et =>)
      Move(in := 2, out1 => "AI SCALING DB"."LT-201".LOW_BUFF)
   END_RUNG
   RUNG wire#w1
      { S7_Templates := "SrcType := Real" } LT_Contact(in1 := "AI SCALING DB".PV."LEVEL TRANSMITTER-201", in2 := "AI SCALING DB"."LT-201 SET VALVE".H)
      { S7_Templates := "time_type := Time" } "IEC_Timer_0_DB_28".TON(pt := T#3S, et =>)
      Move(in := 3, out1 => "AI SCALING DB"."LT-201".HIGH_BUFF)
   END_RUNG
   RUNG wire#w1
      { S7_Templates := "SrcType := Real" } GE_Contact(in1 := "AI SCALING DB".PV."LEVEL TRANSMITTER-201", in2 := "AI SCALING DB"."LT-201 SET VALVE".HH)
      { S7_Templates := "time_type := Time" } "IEC_Timer_0_DB_29".TON(pt := T#3S, et =>)
      Move(in := 4, out1 => "AI SCALING DB"."LT-201".HIGH_BUFF)
   END_RUNG
   RUNG wire#powerrail
      Contact( "AlwaysTRUE" )
      wire#w2
      { S7_Templates := "SrcType := Real" } GE_Contact(in1 := "AI SCALING DB".PV."LEVEL TRANSMITTER-201", in2 := "AI SCALING DB"."LT-201 SET VALVE".LL)
      { S7_Templates := "time_type := Time" } "IEC_Timer_0_DB_91".TON(pt := T#5S, et =>)
      Move(in := 1, out1 => "ONLY_UF BACKWASH LT201 LL")
   END_RUNG
   RUNG wire#w2
      { S7_Templates := "SrcType := Real" } LT_Contact(in1 := "AI SCALING DB".PV."LEVEL TRANSMITTER-201", in2 := "AI SCALING DB"."LT-201 SET VALVE".LL)
      { S7_Templates := "time_type := Time" } "IEC_Timer_0_DB_94".TON(pt := T#5S, et =>)
      Move(in := 0, out1 => "ONLY_UF BACKWASH LT201 LL")
   END_RUNG
   // the same network as SCL:
   "IEC_Timer_0_DB_26".TON(IN := "AlwaysTRUE" AND ("AI SCALING DB".PV."LEVEL TRANSMITTER-201" < "AI SCALING DB"."LT-201 SET VALVE".LL),
                           PT := T#3S);
   IF "IEC_Timer_0_DB_26".Q THEN "AI SCALING DB"."LT-201".LOW_BUFF := 1; END_IF;
   "IEC_Timer_0_DB_27".TON(IN := "AlwaysTRUE" AND ("AI SCALING DB".PV."LEVEL TRANSMITTER-201" >= "AI SCALING DB"."LT-201 SET VALVE".L),
                           PT := T#3S);
   IF "IEC_Timer_0_DB_27".Q THEN "AI SCALING DB"."LT-201".LOW_BUFF := 2; END_IF;
   "IEC_Timer_0_DB_28".TON(IN := "AlwaysTRUE" AND ("AI SCALING DB".PV."LEVEL TRANSMITTER-201" < "AI SCALING DB"."LT-201 SET VALVE".H),
                           PT := T#3S);
   IF "IEC_Timer_0_DB_28".Q THEN "AI SCALING DB"."LT-201".HIGH_BUFF := 3; END_IF;
   "IEC_Timer_0_DB_29".TON(IN := "AlwaysTRUE" AND ("AI SCALING DB".PV."LEVEL TRANSMITTER-201" >= "AI SCALING DB"."LT-201 SET VALVE".HH),
                           PT := T#3S);
   IF "IEC_Timer_0_DB_29".Q THEN "AI SCALING DB"."LT-201".HIGH_BUFF := 4; END_IF;
   "IEC_Timer_0_DB_91".TON(IN := "AlwaysTRUE" AND ("AI SCALING DB".PV."LEVEL TRANSMITTER-201" >= "AI SCALING DB"."LT-201 SET VALVE".LL),
                           PT := T#5S);
   IF "IEC_Timer_0_DB_91".Q THEN "ONLY_UF BACKWASH LT201 LL" := 1; END_IF;
   "IEC_Timer_0_DB_94".TON(IN := "AlwaysTRUE" AND ("AI SCALING DB".PV."LEVEL TRANSMITTER-201" < "AI SCALING DB"."LT-201 SET VALVE".LL),
                           PT := T#5S);
   IF "IEC_Timer_0_DB_94".Q THEN "ONLY_UF BACKWASH LT201 LL" := 0; END_IF;
END_REGION

REGION Network 19: LT-801 BUFFER
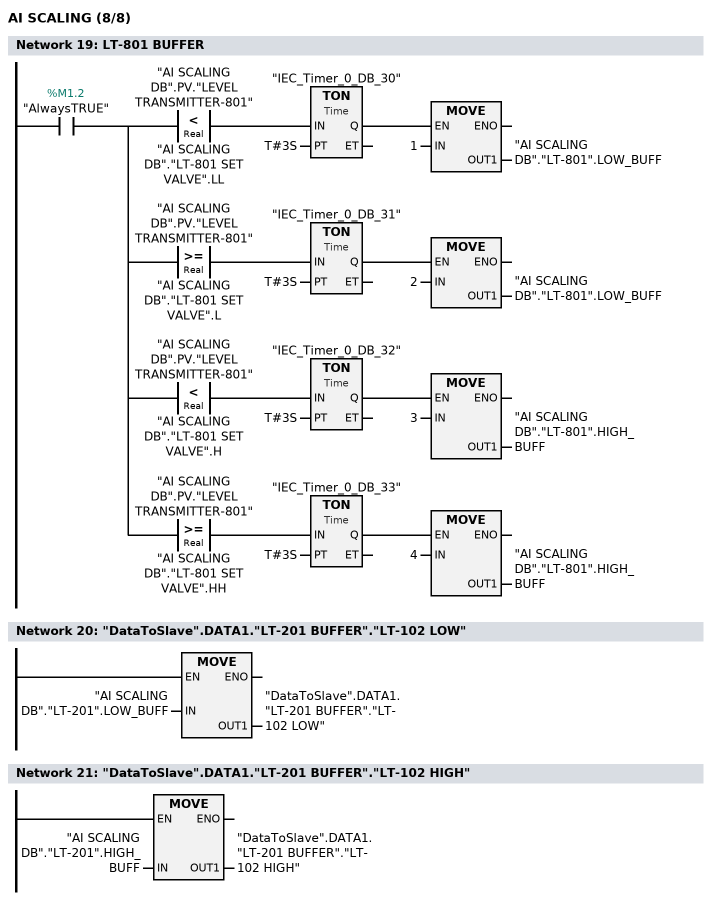
   RUNG wire#powerrail
      Contact( "AlwaysTRUE" )
      wire#w1
      { S7_Templates := "SrcType := Real" } LT_Contact(in1 := "AI SCALING DB".PV."LEVEL TRANSMITTER-801", in2 := "AI SCALING DB"."LT-801 SET VALVE".LL)
      { S7_Templates := "time_type := Time" } "IEC_Timer_0_DB_30".TON(pt := T#3S, et =>)
      Move(in := 1, out1 => "AI SCALING DB"."LT-801".LOW_BUFF)
   END_RUNG
   RUNG wire#w1
      { S7_Templates := "SrcType := Real" } GE_Contact(in1 := "AI SCALING DB".PV."LEVEL TRANSMITTER-801", in2 := "AI SCALING DB"."LT-801 SET VALVE".L)
      { S7_Templates := "time_type := Time" } "IEC_Timer_0_DB_31".TON(pt := T#3S, et =>)
      Move(in := 2, out1 => "AI SCALING DB"."LT-801".LOW_BUFF)
   END_RUNG
   RUNG wire#w1
      { S7_Templates := "SrcType := Real" } LT_Contact(in1 := "AI SCALING DB".PV."LEVEL TRANSMITTER-801", in2 := "AI SCALING DB"."LT-801 SET VALVE".H)
      { S7_Templates := "time_type := Time" } "IEC_Timer_0_DB_32".TON(pt := T#3S, et =>)
      Move(in := 3, out1 => "AI SCALING DB"."LT-801".HIGH_BUFF)
   END_RUNG
   RUNG wire#w1
      { S7_Templates := "SrcType := Real" } GE_Contact(in1 := "AI SCALING DB".PV."LEVEL TRANSMITTER-801", in2 := "AI SCALING DB"."LT-801 SET VALVE".HH)
      { S7_Templates := "time_type := Time" } "IEC_Timer_0_DB_33".TON(pt := T#3S, et =>)
      Move(in := 4, out1 => "AI SCALING DB"."LT-801".HIGH_BUFF)
   END_RUNG
   // the same network as SCL:
   "IEC_Timer_0_DB_30".TON(IN := "AlwaysTRUE" AND ("AI SCALING DB".PV."LEVEL TRANSMITTER-801" < "AI SCALING DB"."LT-801 SET VALVE".LL),
                           PT := T#3S);
   IF "IEC_Timer_0_DB_30".Q THEN "AI SCALING DB"."LT-801".LOW_BUFF := 1; END_IF;
   "IEC_Timer_0_DB_31".TON(IN := "AlwaysTRUE" AND ("AI SCALING DB".PV."LEVEL TRANSMITTER-801" >= "AI SCALING DB"."LT-801 SET VALVE".L),
                           PT := T#3S);
   IF "IEC_Timer_0_DB_31".Q THEN "AI SCALING DB"."LT-801".LOW_BUFF := 2; END_IF;
   "IEC_Timer_0_DB_32".TON(IN := "AlwaysTRUE" AND ("AI SCALING DB".PV."LEVEL TRANSMITTER-801" < "AI SCALING DB"."LT-801 SET VALVE".H),
                           PT := T#3S);
   IF "IEC_Timer_0_DB_32".Q THEN "AI SCALING DB"."LT-801".HIGH_BUFF := 3; END_IF;
   "IEC_Timer_0_DB_33".TON(IN := "AlwaysTRUE" AND ("AI SCALING DB".PV."LEVEL TRANSMITTER-801" >= "AI SCALING DB"."LT-801 SET VALVE".HH),
                           PT := T#3S);
   IF "IEC_Timer_0_DB_33".Q THEN "AI SCALING DB"."LT-801".HIGH_BUFF := 4; END_IF;
END_REGION

REGION Network 20: "DataToSlave".DATA1."LT-201 BUFFER"."LT-102 LOW"
   RUNG wire#powerrail
      Move(in := "AI SCALING DB"."LT-201".LOW_BUFF, out1 => "DataToSlave".DATA1."LT-201 BUFFER"."LT-102 LOW")
   END_RUNG
   // the same network as SCL:
   "DataToSlave".DATA1."LT-201 BUFFER"."LT-102 LOW" := "AI SCALING DB"."LT-201".LOW_BUFF;
END_REGION

REGION Network 21: "DataToSlave".DATA1."LT-201 BUFFER"."LT-102 HIGH"
   RUNG wire#powerrail
      Move(in := "AI SCALING DB"."LT-201".HIGH_BUFF, out1 => "DataToSlave".DATA1."LT-201 BUFFER"."LT-102 HIGH")
   END_RUNG
   // the same network as SCL:
   "DataToSlave".DATA1."LT-201 BUFFER"."LT-102 HIGH" := "AI SCALING DB"."LT-201".HIGH_BUFF;
END_REGION
END_FUNCTION

FUNCTION "INPUT MAPPING" : Void   // FC3, LAD
{ S7_Optimized_Access := 'TRUE' }
// stored: SetENOAutomatically false
BEGIN

REGION Network 1: EMERGENCY STOP
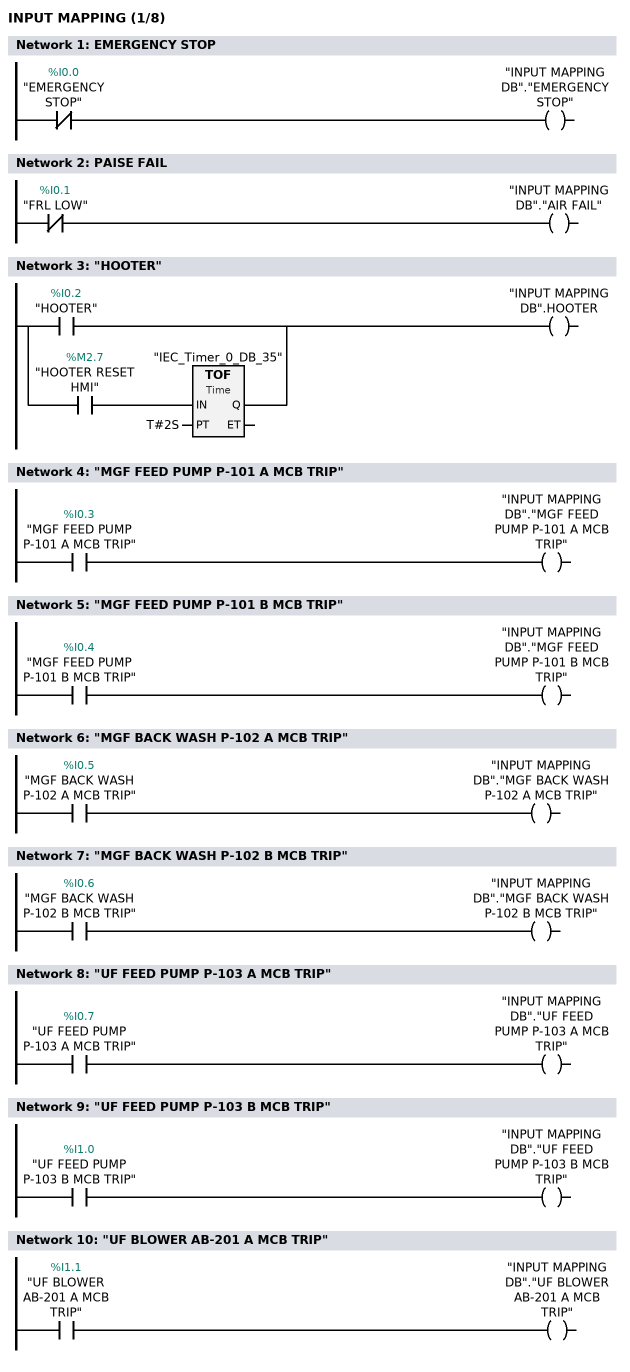
   RUNG wire#powerrail
      I_Contact( "EMERGENCY STOP" )
      Coil( "INPUT MAPPING DB"."EMERGENCY STOP" )
   END_RUNG
   // the same network as SCL:
   "INPUT MAPPING DB"."EMERGENCY STOP" := NOT "EMERGENCY STOP";
END_REGION

REGION Network 2: PAISE FAIL
   RUNG wire#powerrail
      I_Contact( "FRL LOW" )
      Coil( "INPUT MAPPING DB"."AIR FAIL" )
   END_RUNG
   // the same network as SCL:
   "INPUT MAPPING DB"."AIR FAIL" := NOT "FRL LOW";
END_REGION

REGION Network 3: "HOOTER"
   RUNG wire#powerrail
      Contact( "HOOTER" )
      wire#w1
      Coil( "INPUT MAPPING DB".HOOTER )
   END_RUNG
   RUNG wire#powerrail
      Contact( "HOOTER RESET HMI" )
      { S7_Templates := "time_type := Time" } "IEC_Timer_0_DB_35".TOF(pt := T#2S, et =>)
   END_RUNG wire#w1
   // the same network as SCL:
   "IEC_Timer_0_DB_35".TOF(IN := "HOOTER RESET HMI", PT := T#2S);
   "INPUT MAPPING DB".HOOTER := "HOOTER" OR "IEC_Timer_0_DB_35".Q;
END_REGION

REGION Network 4: "MGF FEED PUMP P-101 A MCB TRIP"
   RUNG wire#powerrail
      Contact( "MGF FEED PUMP P-101 A MCB TRIP" )
      Coil( "INPUT MAPPING DB"."MGF FEED PUMP P-101 A MCB TRIP" )
   END_RUNG
   // the same network as SCL:
   "INPUT MAPPING DB"."MGF FEED PUMP P-101 A MCB TRIP" := "MGF FEED PUMP P-101 A MCB TRIP";
END_REGION

REGION Network 5: "MGF FEED PUMP P-101 B MCB TRIP"
   RUNG wire#powerrail
      Contact( "MGF FEED PUMP P-101 B MCB TRIP" )
      Coil( "INPUT MAPPING DB"."MGF FEED PUMP P-101 B MCB TRIP" )
   END_RUNG
   // the same network as SCL:
   "INPUT MAPPING DB"."MGF FEED PUMP P-101 B MCB TRIP" := "MGF FEED PUMP P-101 B MCB TRIP";
END_REGION

REGION Network 6: "MGF BACK WASH P-102 A MCB TRIP"
   RUNG wire#powerrail
      Contact( "MGF BACK WASH  P-102 A MCB TRIP" )
      Coil( "INPUT MAPPING DB"."MGF BACK WASH  P-102 A MCB TRIP" )
   END_RUNG
   // the same network as SCL:
   "INPUT MAPPING DB"."MGF BACK WASH  P-102 A MCB TRIP" := "MGF BACK WASH  P-102 A MCB TRIP";
END_REGION

REGION Network 7: "MGF BACK WASH P-102 B MCB TRIP"
   RUNG wire#powerrail
      Contact( "MGF BACK WASH P-102 B MCB TRIP" )
      Coil( "INPUT MAPPING DB"."MGF BACK WASH P-102 B MCB TRIP" )
   END_RUNG
   // the same network as SCL:
   "INPUT MAPPING DB"."MGF BACK WASH P-102 B MCB TRIP" := "MGF BACK WASH P-102 B MCB TRIP";
END_REGION

REGION Network 8: "UF FEED PUMP P-103 A MCB TRIP"
   RUNG wire#powerrail
      Contact( "UF FEED PUMP P-103 A MCB TRIP" )
      Coil( "INPUT MAPPING DB"."UF FEED PUMP P-103 A MCB TRIP" )
   END_RUNG
   // the same network as SCL:
   "INPUT MAPPING DB"."UF FEED PUMP P-103 A MCB TRIP" := "UF FEED PUMP P-103 A MCB TRIP";
END_REGION

REGION Network 9: "UF FEED PUMP P-103 B MCB TRIP"
   RUNG wire#powerrail
      Contact( "UF FEED PUMP P-103 B MCB TRIP" )
      Coil( "INPUT MAPPING DB"."UF FEED PUMP P-103 B MCB TRIP" )
   END_RUNG
   // the same network as SCL:
   "INPUT MAPPING DB"."UF FEED PUMP P-103 B MCB TRIP" := "UF FEED PUMP P-103 B MCB TRIP";
END_REGION

REGION Network 10: "UF BLOWER AB-201 A MCB TRIP"
   RUNG wire#powerrail
      Contact( "UF BLOWER AB-201 A MCB TRIP" )
      Coil( "INPUT MAPPING DB"."UF BLOWER AB-201 A MCB TRIP" )
   END_RUNG
   // the same network as SCL:
   "INPUT MAPPING DB"."UF BLOWER AB-201 A MCB TRIP" := "UF BLOWER AB-201 A MCB TRIP";
END_REGION

REGION Network 11: "UF BLOWER AB-201 B MCB TRIP"
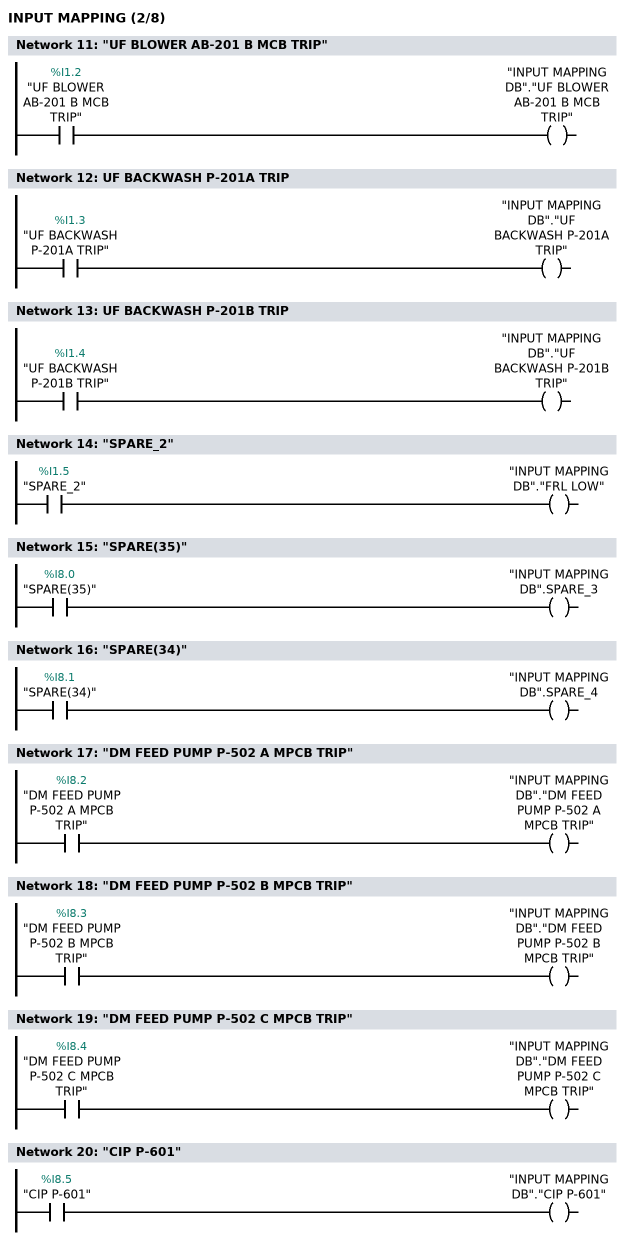
   RUNG wire#powerrail
      Contact( "UF BLOWER AB-201 B MCB TRIP" )
      Coil( "INPUT MAPPING DB"."UF BLOWER AB-201 B MCB TRIP" )
   END_RUNG
   // the same network as SCL:
   "INPUT MAPPING DB"."UF BLOWER AB-201 B MCB TRIP" := "UF BLOWER AB-201 B MCB TRIP";
END_REGION

REGION Network 12: UF BACKWASH P-201A TRIP
   RUNG wire#powerrail
      Contact( "UF BACKWASH P-201A TRIP" )
      Coil( "INPUT MAPPING DB"."UF BACKWASH P-201A TRIP" )
   END_RUNG
   // the same network as SCL:
   "INPUT MAPPING DB"."UF BACKWASH P-201A TRIP" := "UF BACKWASH P-201A TRIP";
END_REGION

REGION Network 13: UF BACKWASH P-201B TRIP
   RUNG wire#powerrail
      Contact( "UF BACKWASH P-201B TRIP" )
      Coil( "INPUT MAPPING DB"."UF BACKWASH P-201B TRIP" )
   END_RUNG
   // the same network as SCL:
   "INPUT MAPPING DB"."UF BACKWASH P-201B TRIP" := "UF BACKWASH P-201B TRIP";
END_REGION

REGION Network 14: "SPARE_2"
   RUNG wire#powerrail
      Contact( "SPARE_2" )
      Coil( "INPUT MAPPING DB"."FRL LOW" )
   END_RUNG
   // the same network as SCL:
   "INPUT MAPPING DB"."FRL LOW" := "SPARE_2";
END_REGION

REGION Network 15: "SPARE(35)"
   RUNG wire#powerrail
      Contact( "SPARE(35)" )
      Coil( "INPUT MAPPING DB".SPARE_3 )
   END_RUNG
   // the same network as SCL:
   "INPUT MAPPING DB".SPARE_3 := "SPARE(35)";
END_REGION

REGION Network 16: "SPARE(34)"
   RUNG wire#powerrail
      Contact( "SPARE(34)" )
      Coil( "INPUT MAPPING DB".SPARE_4 )
   END_RUNG
   // the same network as SCL:
   "INPUT MAPPING DB".SPARE_4 := "SPARE(34)";
END_REGION

REGION Network 17: "DM FEED PUMP P-502 A MPCB TRIP"
   RUNG wire#powerrail
      Contact( "DM FEED PUMP P-502 A MPCB TRIP" )
      Coil( "INPUT MAPPING DB"."DM FEED PUMP P-502 A MPCB TRIP" )
   END_RUNG
   // the same network as SCL:
   "INPUT MAPPING DB"."DM FEED PUMP P-502 A MPCB TRIP" := "DM FEED PUMP P-502 A MPCB TRIP";
END_REGION

REGION Network 18: "DM FEED PUMP P-502 B MPCB TRIP"
   RUNG wire#powerrail
      Contact( "DM FEED PUMP P-502 B MPCB TRIP" )
      Coil( "INPUT MAPPING DB"."DM FEED PUMP P-502 B MPCB TRIP" )
   END_RUNG
   // the same network as SCL:
   "INPUT MAPPING DB"."DM FEED PUMP P-502 B MPCB TRIP" := "DM FEED PUMP P-502 B MPCB TRIP";
END_REGION

REGION Network 19: "DM FEED PUMP P-502 C MPCB TRIP"
   RUNG wire#powerrail
      Contact( "DM FEED PUMP P-502 C MPCB TRIP" )
      Coil( "INPUT MAPPING DB"."DM FEED PUMP P-502 C MPCB TRIP" )
   END_RUNG
   // the same network as SCL:
   "INPUT MAPPING DB"."DM FEED PUMP P-502 C MPCB TRIP" := "DM FEED PUMP P-502 C MPCB TRIP";
END_REGION

REGION Network 20: "CIP P-601"
   RUNG wire#powerrail
      Contact( "CIP P-601" )
      Coil( "INPUT MAPPING DB"."CIP P-601" )
   END_RUNG
   // the same network as SCL:
   "INPUT MAPPING DB"."CIP P-601" := "CIP P-601";
END_REGION

REGION Network 21: "BACK WASH RECOVERY P-801 A MPCB TRIP"
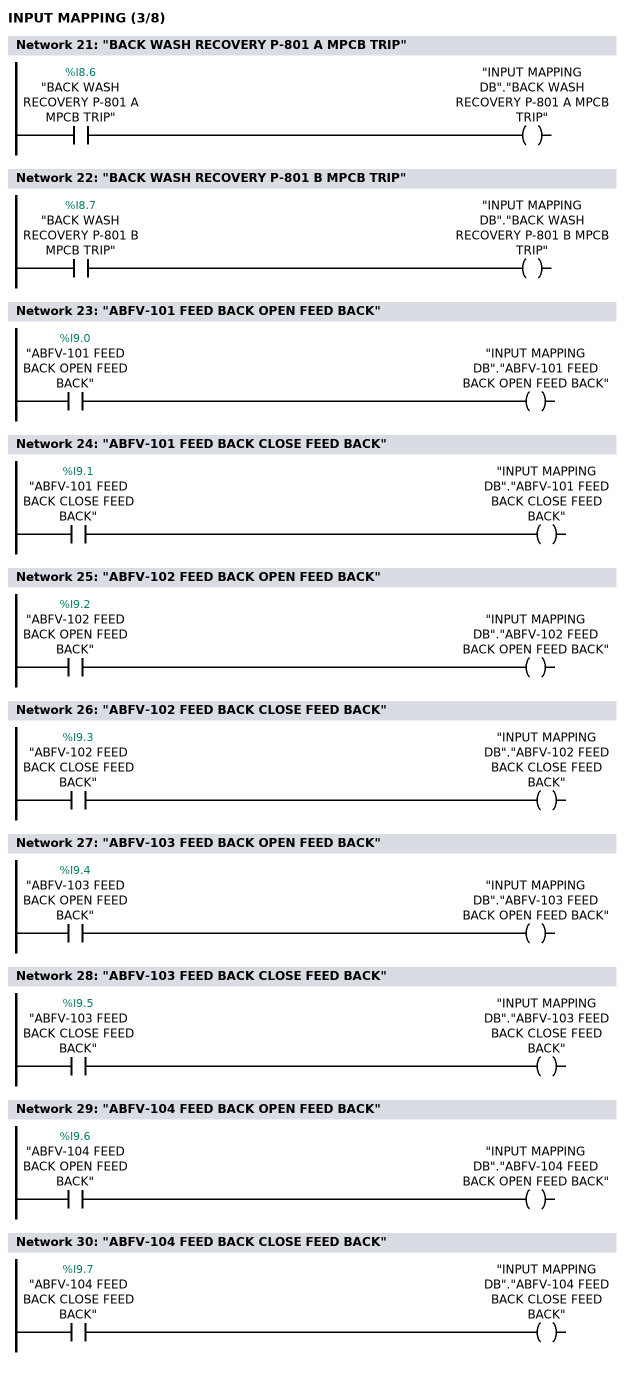
   RUNG wire#powerrail
      Contact( "BACK WASH RECOVERY P-801 A MPCB TRIP" )
      Coil( "INPUT MAPPING DB"."BACK WASH RECOVERY P-801 A MPCB TRIP" )
   END_RUNG
   // the same network as SCL:
   "INPUT MAPPING DB"."BACK WASH RECOVERY P-801 A MPCB TRIP" := "BACK WASH RECOVERY P-801 A MPCB TRIP";
END_REGION

REGION Network 22: "BACK WASH RECOVERY P-801 B MPCB TRIP"
   RUNG wire#powerrail
      Contact( "BACK WASH RECOVERY P-801 B MPCB TRIP" )
      Coil( "INPUT MAPPING DB"."BACK WASH RECOVERY P-801 B MPCB TRIP" )
   END_RUNG
   // the same network as SCL:
   "INPUT MAPPING DB"."BACK WASH RECOVERY P-801 B MPCB TRIP" := "BACK WASH RECOVERY P-801 B MPCB TRIP";
END_REGION

REGION Network 23: "ABFV-101 FEED BACK OPEN FEED BACK"
   RUNG wire#powerrail
      Contact( "ABFV-101 FEED BACK OPEN FEED BACK" )
      Coil( "INPUT MAPPING DB"."ABFV-101 FEED BACK OPEN FEED BACK" )
   END_RUNG
   // the same network as SCL:
   "INPUT MAPPING DB"."ABFV-101 FEED BACK OPEN FEED BACK" := "ABFV-101 FEED BACK OPEN FEED BACK";
END_REGION

REGION Network 24: "ABFV-101 FEED BACK CLOSE FEED BACK"
   RUNG wire#powerrail
      Contact( "ABFV-101 FEED BACK CLOSE FEED BACK" )
      Coil( "INPUT MAPPING DB"."ABFV-101 FEED BACK CLOSE FEED BACK" )
   END_RUNG
   // the same network as SCL:
   "INPUT MAPPING DB"."ABFV-101 FEED BACK CLOSE FEED BACK" := "ABFV-101 FEED BACK CLOSE FEED BACK";
END_REGION

REGION Network 25: "ABFV-102 FEED BACK OPEN FEED BACK"
   RUNG wire#powerrail
      Contact( "ABFV-102 FEED BACK OPEN FEED BACK" )
      Coil( "INPUT MAPPING DB"."ABFV-102 FEED BACK OPEN FEED BACK" )
   END_RUNG
   // the same network as SCL:
   "INPUT MAPPING DB"."ABFV-102 FEED BACK OPEN FEED BACK" := "ABFV-102 FEED BACK OPEN FEED BACK";
END_REGION

REGION Network 26: "ABFV-102 FEED BACK CLOSE FEED BACK"
   RUNG wire#powerrail
      Contact( "ABFV-102 FEED BACK CLOSE FEED BACK" )
      Coil( "INPUT MAPPING DB"."ABFV-102 FEED BACK CLOSE FEED BACK" )
   END_RUNG
   // the same network as SCL:
   "INPUT MAPPING DB"."ABFV-102 FEED BACK CLOSE FEED BACK" := "ABFV-102 FEED BACK CLOSE FEED BACK";
END_REGION

REGION Network 27: "ABFV-103 FEED BACK OPEN FEED BACK"
   RUNG wire#powerrail
      Contact( "ABFV-103 FEED BACK OPEN FEED BACK" )
      Coil( "INPUT MAPPING DB"."ABFV-103 FEED BACK OPEN FEED BACK" )
   END_RUNG
   // the same network as SCL:
   "INPUT MAPPING DB"."ABFV-103 FEED BACK OPEN FEED BACK" := "ABFV-103 FEED BACK OPEN FEED BACK";
END_REGION

REGION Network 28: "ABFV-103 FEED BACK CLOSE FEED BACK"
   RUNG wire#powerrail
      Contact( "ABFV-103 FEED BACK CLOSE FEED BACK" )
      Coil( "INPUT MAPPING DB"."ABFV-103 FEED BACK CLOSE FEED BACK" )
   END_RUNG
   // the same network as SCL:
   "INPUT MAPPING DB"."ABFV-103 FEED BACK CLOSE FEED BACK" := "ABFV-103 FEED BACK CLOSE FEED BACK";
END_REGION

REGION Network 29: "ABFV-104 FEED BACK OPEN FEED BACK"
   RUNG wire#powerrail
      Contact( "ABFV-104 FEED BACK OPEN FEED BACK" )
      Coil( "INPUT MAPPING DB"."ABFV-104 FEED BACK OPEN FEED BACK" )
   END_RUNG
   // the same network as SCL:
   "INPUT MAPPING DB"."ABFV-104 FEED BACK OPEN FEED BACK" := "ABFV-104 FEED BACK OPEN FEED BACK";
END_REGION

REGION Network 30: "ABFV-104 FEED BACK CLOSE FEED BACK"
   RUNG wire#powerrail
      Contact( "ABFV-104 FEED BACK CLOSE FEED BACK" )
      Coil( "INPUT MAPPING DB"."ABFV-104 FEED BACK CLOSE FEED BACK" )
   END_RUNG
   // the same network as SCL:
   "INPUT MAPPING DB"."ABFV-104 FEED BACK CLOSE FEED BACK" := "ABFV-104 FEED BACK CLOSE FEED BACK";
END_REGION

REGION Network 31: "ABFV 105 FEED BACK OPEN"
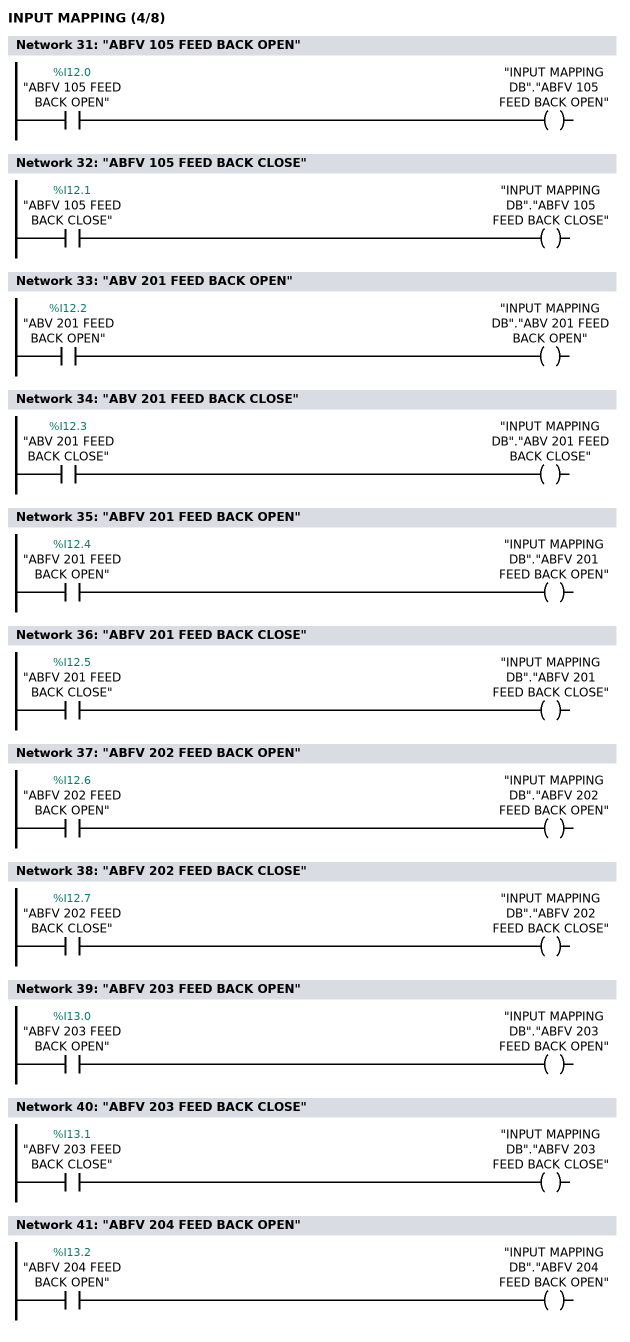
   RUNG wire#powerrail
      Contact( "ABFV 105 FEED BACK OPEN" )
      Coil( "INPUT MAPPING DB"."ABFV 105 FEED BACK OPEN" )
   END_RUNG
   // the same network as SCL:
   "INPUT MAPPING DB"."ABFV 105 FEED BACK OPEN" := "ABFV 105 FEED BACK OPEN";
END_REGION

REGION Network 32: "ABFV 105 FEED BACK CLOSE"
   RUNG wire#powerrail
      Contact( "ABFV 105 FEED BACK CLOSE" )
      Coil( "INPUT MAPPING DB"."ABFV 105 FEED BACK CLOSE" )
   END_RUNG
   // the same network as SCL:
   "INPUT MAPPING DB"."ABFV 105 FEED BACK CLOSE" := "ABFV 105 FEED BACK CLOSE";
END_REGION

REGION Network 33: "ABV 201 FEED BACK OPEN"
   RUNG wire#powerrail
      Contact( "ABV 201 FEED BACK OPEN" )
      Coil( "INPUT MAPPING DB"."ABV 201 FEED BACK OPEN" )
   END_RUNG
   // the same network as SCL:
   "INPUT MAPPING DB"."ABV 201 FEED BACK OPEN" := "ABV 201 FEED BACK OPEN";
END_REGION

REGION Network 34: "ABV 201 FEED BACK CLOSE"
   RUNG wire#powerrail
      Contact( "ABV 201 FEED BACK CLOSE" )
      Coil( "INPUT MAPPING DB"."ABV 201 FEED BACK CLOSE" )
   END_RUNG
   // the same network as SCL:
   "INPUT MAPPING DB"."ABV 201 FEED BACK CLOSE" := "ABV 201 FEED BACK CLOSE";
END_REGION

REGION Network 35: "ABFV 201 FEED BACK OPEN"
   RUNG wire#powerrail
      Contact( "ABFV 201 FEED BACK OPEN" )
      Coil( "INPUT MAPPING DB"."ABFV 201 FEED BACK OPEN" )
   END_RUNG
   // the same network as SCL:
   "INPUT MAPPING DB"."ABFV 201 FEED BACK OPEN" := "ABFV 201 FEED BACK OPEN";
END_REGION

REGION Network 36: "ABFV 201 FEED BACK CLOSE"
   RUNG wire#powerrail
      Contact( "ABFV 201 FEED BACK CLOSE" )
      Coil( "INPUT MAPPING DB"."ABFV 201 FEED BACK CLOSE" )
   END_RUNG
   // the same network as SCL:
   "INPUT MAPPING DB"."ABFV 201 FEED BACK CLOSE" := "ABFV 201 FEED BACK CLOSE";
END_REGION

REGION Network 37: "ABFV 202 FEED BACK OPEN"
   RUNG wire#powerrail
      Contact( "ABFV 202 FEED BACK OPEN" )
      Coil( "INPUT MAPPING DB"."ABFV 202 FEED BACK OPEN" )
   END_RUNG
   // the same network as SCL:
   "INPUT MAPPING DB"."ABFV 202 FEED BACK OPEN" := "ABFV 202 FEED BACK OPEN";
END_REGION

REGION Network 38: "ABFV 202 FEED BACK CLOSE"
   RUNG wire#powerrail
      Contact( "ABFV 202 FEED BACK CLOSE" )
      Coil( "INPUT MAPPING DB"."ABFV 202 FEED BACK CLOSE" )
   END_RUNG
   // the same network as SCL:
   "INPUT MAPPING DB"."ABFV 202 FEED BACK CLOSE" := "ABFV 202 FEED BACK CLOSE";
END_REGION

REGION Network 39: "ABFV 203 FEED BACK OPEN"
   RUNG wire#powerrail
      Contact( "ABFV 203 FEED BACK OPEN" )
      Coil( "INPUT MAPPING DB"."ABFV 203 FEED BACK OPEN" )
   END_RUNG
   // the same network as SCL:
   "INPUT MAPPING DB"."ABFV 203 FEED BACK OPEN" := "ABFV 203 FEED BACK OPEN";
END_REGION

REGION Network 40: "ABFV 203 FEED BACK CLOSE"
   RUNG wire#powerrail
      Contact( "ABFV 203 FEED BACK CLOSE" )
      Coil( "INPUT MAPPING DB"."ABFV 203 FEED BACK CLOSE" )
   END_RUNG
   // the same network as SCL:
   "INPUT MAPPING DB"."ABFV 203 FEED BACK CLOSE" := "ABFV 203 FEED BACK CLOSE";
END_REGION

REGION Network 41: "ABFV 204 FEED BACK OPEN"
   RUNG wire#powerrail
      Contact( "ABFV 204 FEED BACK OPEN" )
      Coil( "INPUT MAPPING DB"."ABFV 204 FEED BACK OPEN" )
   END_RUNG
   // the same network as SCL:
   "INPUT MAPPING DB"."ABFV 204 FEED BACK OPEN" := "ABFV 204 FEED BACK OPEN";
END_REGION

REGION Network 42: "ABFV 204 FEED BACK CLOSE"
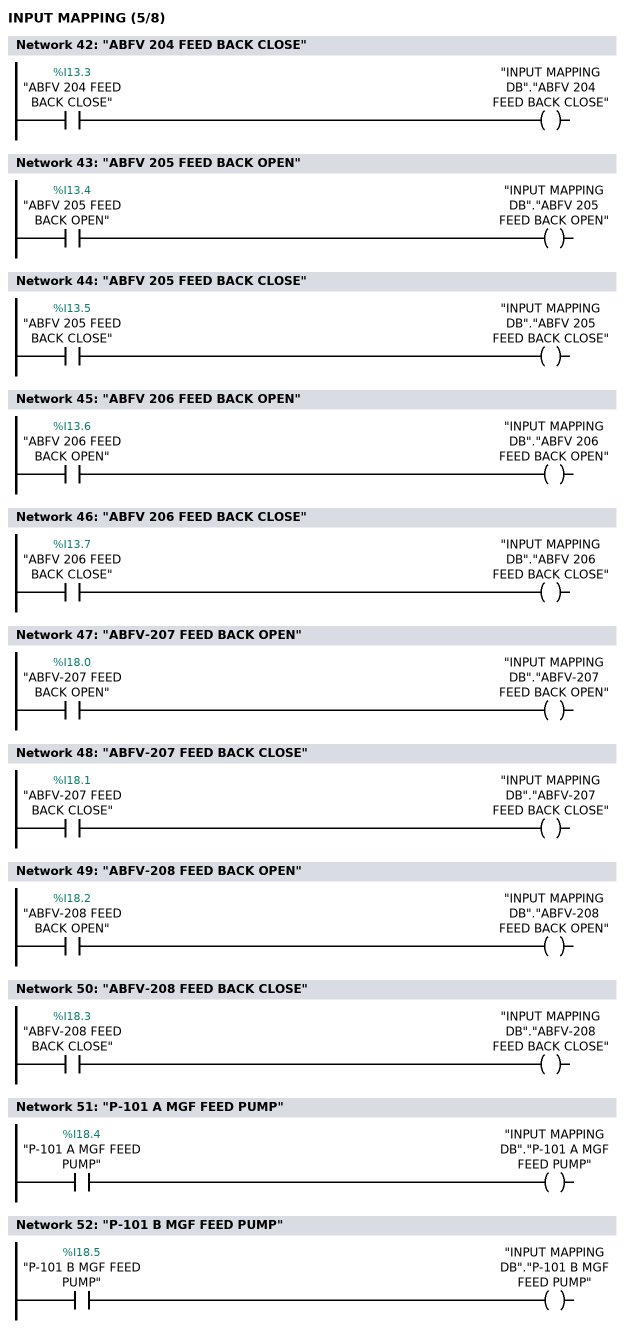
   RUNG wire#powerrail
      Contact( "ABFV 204 FEED BACK CLOSE" )
      Coil( "INPUT MAPPING DB"."ABFV 204 FEED BACK CLOSE" )
   END_RUNG
   // the same network as SCL:
   "INPUT MAPPING DB"."ABFV 204 FEED BACK CLOSE" := "ABFV 204 FEED BACK CLOSE";
END_REGION

REGION Network 43: "ABFV 205 FEED BACK OPEN"
   RUNG wire#powerrail
      Contact( "ABFV 205 FEED BACK OPEN" )
      Coil( "INPUT MAPPING DB"."ABFV 205 FEED BACK OPEN" )
   END_RUNG
   // the same network as SCL:
   "INPUT MAPPING DB"."ABFV 205 FEED BACK OPEN" := "ABFV 205 FEED BACK OPEN";
END_REGION

REGION Network 44: "ABFV 205 FEED BACK CLOSE"
   RUNG wire#powerrail
      Contact( "ABFV 205 FEED BACK CLOSE" )
      Coil( "INPUT MAPPING DB"."ABFV 205 FEED BACK CLOSE" )
   END_RUNG
   // the same network as SCL:
   "INPUT MAPPING DB"."ABFV 205 FEED BACK CLOSE" := "ABFV 205 FEED BACK CLOSE";
END_REGION

REGION Network 45: "ABFV 206 FEED BACK OPEN"
   RUNG wire#powerrail
      Contact( "ABFV 206 FEED BACK OPEN" )
      Coil( "INPUT MAPPING DB"."ABFV 206 FEED BACK OPEN" )
   END_RUNG
   // the same network as SCL:
   "INPUT MAPPING DB"."ABFV 206 FEED BACK OPEN" := "ABFV 206 FEED BACK OPEN";
END_REGION

REGION Network 46: "ABFV 206 FEED BACK CLOSE"
   RUNG wire#powerrail
      Contact( "ABFV 206 FEED BACK CLOSE" )
      Coil( "INPUT MAPPING DB"."ABFV 206 FEED BACK CLOSE" )
   END_RUNG
   // the same network as SCL:
   "INPUT MAPPING DB"."ABFV 206 FEED BACK CLOSE" := "ABFV 206 FEED BACK CLOSE";
END_REGION

REGION Network 47: "ABFV-207 FEED BACK OPEN"
   RUNG wire#powerrail
      Contact( "ABFV-207 FEED BACK OPEN" )
      Coil( "INPUT MAPPING DB"."ABFV-207 FEED BACK OPEN" )
   END_RUNG
   // the same network as SCL:
   "INPUT MAPPING DB"."ABFV-207 FEED BACK OPEN" := "ABFV-207 FEED BACK OPEN";
END_REGION

REGION Network 48: "ABFV-207 FEED BACK CLOSE"
   RUNG wire#powerrail
      Contact( "ABFV-207 FEED BACK CLOSE" )
      Coil( "INPUT MAPPING DB"."ABFV-207 FEED BACK CLOSE" )
   END_RUNG
   // the same network as SCL:
   "INPUT MAPPING DB"."ABFV-207 FEED BACK CLOSE" := "ABFV-207 FEED BACK CLOSE";
END_REGION

REGION Network 49: "ABFV-208 FEED BACK OPEN"
   RUNG wire#powerrail
      Contact( "ABFV-208 FEED BACK OPEN" )
      Coil( "INPUT MAPPING DB"."ABFV-208 FEED BACK OPEN" )
   END_RUNG
   // the same network as SCL:
   "INPUT MAPPING DB"."ABFV-208 FEED BACK OPEN" := "ABFV-208 FEED BACK OPEN";
END_REGION

REGION Network 50: "ABFV-208 FEED BACK CLOSE"
   RUNG wire#powerrail
      Contact( "ABFV-208 FEED BACK CLOSE" )
      Coil( "INPUT MAPPING DB"."ABFV-208 FEED BACK CLOSE" )
   END_RUNG
   // the same network as SCL:
   "INPUT MAPPING DB"."ABFV-208 FEED BACK CLOSE" := "ABFV-208 FEED BACK CLOSE";
END_REGION

REGION Network 51: "P-101 A MGF FEED PUMP"
   RUNG wire#powerrail
      Contact( "P-101 A MGF FEED PUMP" )
      Coil( "INPUT MAPPING DB"."P-101 A MGF FEED PUMP" )
   END_RUNG
   // the same network as SCL:
   "INPUT MAPPING DB"."P-101 A MGF FEED PUMP" := "P-101 A MGF FEED PUMP";
END_REGION

REGION Network 52: "P-101 B MGF FEED PUMP"
   RUNG wire#powerrail
      Contact( "P-101 B MGF FEED PUMP" )
      Coil( "INPUT MAPPING DB"."P-101 B MGF FEED PUMP" )
   END_RUNG
   // the same network as SCL:
   "INPUT MAPPING DB"."P-101 B MGF FEED PUMP" := "P-101 B MGF FEED PUMP";
END_REGION

REGION Network 53: "P-102 A MGF BACK WASH"
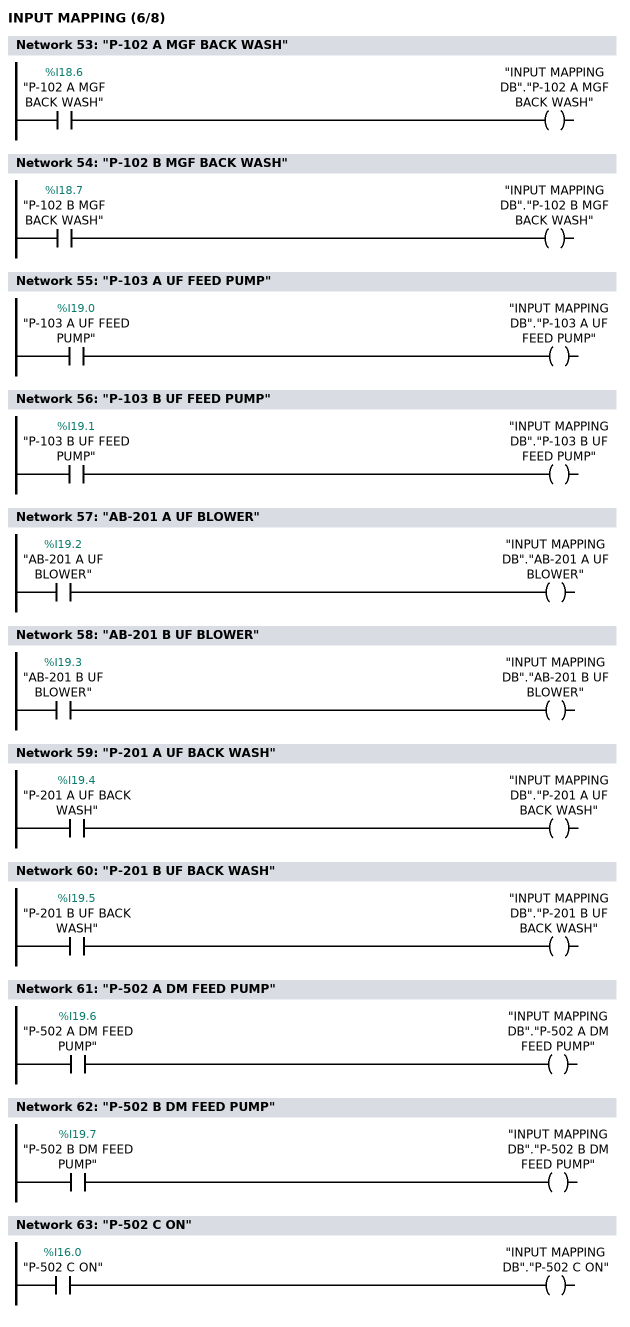
   RUNG wire#powerrail
      Contact( "P-102 A MGF BACK WASH" )
      Coil( "INPUT MAPPING DB"."P-102 A MGF BACK WASH" )
   END_RUNG
   // the same network as SCL:
   "INPUT MAPPING DB"."P-102 A MGF BACK WASH" := "P-102 A MGF BACK WASH";
END_REGION

REGION Network 54: "P-102 B MGF BACK WASH"
   RUNG wire#powerrail
      Contact( "P-102 B MGF BACK WASH" )
      Coil( "INPUT MAPPING DB"."P-102 B MGF BACK WASH" )
   END_RUNG
   // the same network as SCL:
   "INPUT MAPPING DB"."P-102 B MGF BACK WASH" := "P-102 B MGF BACK WASH";
END_REGION

REGION Network 55: "P-103 A UF FEED PUMP"
   RUNG wire#powerrail
      Contact( "P-103 A UF FEED PUMP" )
      Coil( "INPUT MAPPING DB"."P-103 A UF FEED PUMP" )
   END_RUNG
   // the same network as SCL:
   "INPUT MAPPING DB"."P-103 A UF FEED PUMP" := "P-103 A UF FEED PUMP";
END_REGION

REGION Network 56: "P-103 B UF FEED PUMP"
   RUNG wire#powerrail
      Contact( "P-103 B UF FEED PUMP" )
      Coil( "INPUT MAPPING DB"."P-103 B UF FEED PUMP" )
   END_RUNG
   // the same network as SCL:
   "INPUT MAPPING DB"."P-103 B UF FEED PUMP" := "P-103 B UF FEED PUMP";
END_REGION

REGION Network 57: "AB-201 A UF BLOWER"
   RUNG wire#powerrail
      Contact( "AB-201 A UF BLOWER" )
      Coil( "INPUT MAPPING DB"."AB-201 A UF BLOWER" )
   END_RUNG
   // the same network as SCL:
   "INPUT MAPPING DB"."AB-201 A UF BLOWER" := "AB-201 A UF BLOWER";
END_REGION

REGION Network 58: "AB-201 B UF BLOWER"
   RUNG wire#powerrail
      Contact( "AB-201 B UF BLOWER" )
      Coil( "INPUT MAPPING DB"."AB-201 B UF BLOWER" )
   END_RUNG
   // the same network as SCL:
   "INPUT MAPPING DB"."AB-201 B UF BLOWER" := "AB-201 B UF BLOWER";
END_REGION

REGION Network 59: "P-201 A UF BACK WASH"
   RUNG wire#powerrail
      Contact( "P-201 A UF BACK WASH" )
      Coil( "INPUT MAPPING DB"."P-201 A UF BACK WASH" )
   END_RUNG
   // the same network as SCL:
   "INPUT MAPPING DB"."P-201 A UF BACK WASH" := "P-201 A UF BACK WASH";
END_REGION

REGION Network 60: "P-201 B UF BACK WASH"
   RUNG wire#powerrail
      Contact( "P-201 B UF BACK WASH" )
      Coil( "INPUT MAPPING DB"."P-201 B UF BACK WASH" )
   END_RUNG
   // the same network as SCL:
   "INPUT MAPPING DB"."P-201 B UF BACK WASH" := "P-201 B UF BACK WASH";
END_REGION

REGION Network 61: "P-502 A DM FEED PUMP"
   RUNG wire#powerrail
      Contact( "P-502 A DM FEED PUMP" )
      Coil( "INPUT MAPPING DB"."P-502 A DM FEED PUMP" )
   END_RUNG
   // the same network as SCL:
   "INPUT MAPPING DB"."P-502 A DM FEED PUMP" := "P-502 A DM FEED PUMP";
END_REGION

REGION Network 62: "P-502 B DM FEED PUMP"
   RUNG wire#powerrail
      Contact( "P-502 B DM FEED PUMP" )
      Coil( "INPUT MAPPING DB"."P-502 B DM FEED PUMP" )
   END_RUNG
   // the same network as SCL:
   "INPUT MAPPING DB"."P-502 B DM FEED PUMP" := "P-502 B DM FEED PUMP";
END_REGION

REGION Network 63: "P-502 C ON"
   RUNG wire#powerrail
      Contact( "P-502 C ON" )
      Coil( "INPUT MAPPING DB"."P-502 C ON" )
   END_RUNG
   // the same network as SCL:
   "INPUT MAPPING DB"."P-502 C ON" := "P-502 C ON";
END_REGION

REGION Network 64: "P-601 ON"
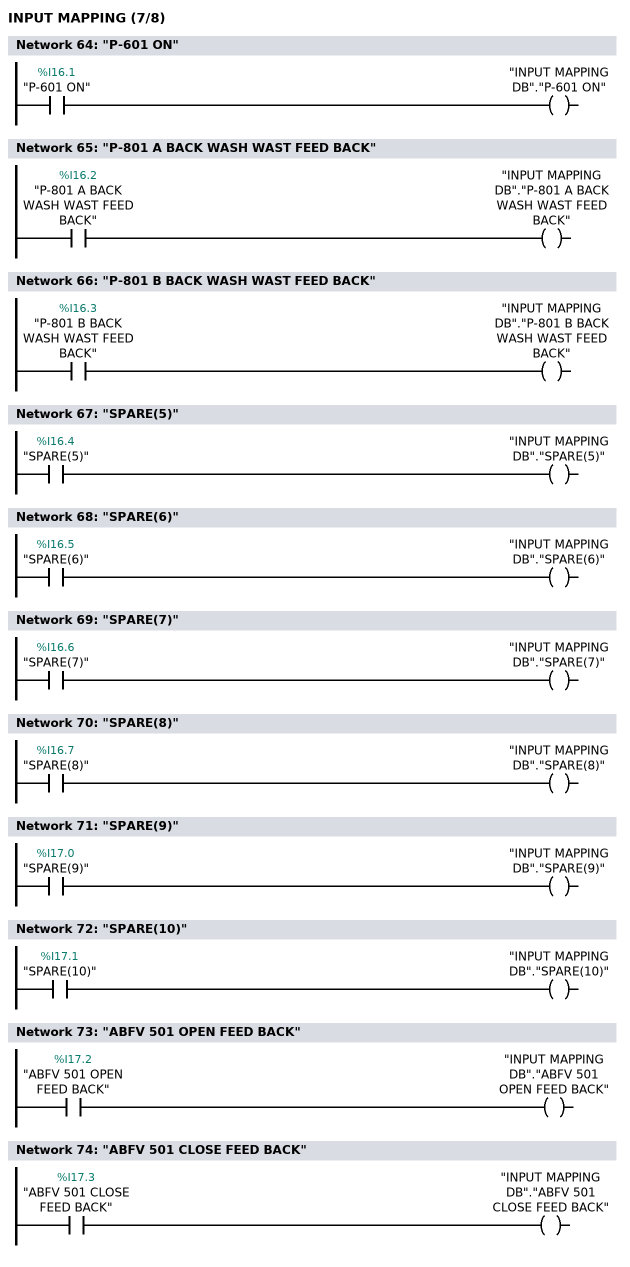
   RUNG wire#powerrail
      Contact( "P-601 ON" )
      Coil( "INPUT MAPPING DB"."P-601 ON" )
   END_RUNG
   // the same network as SCL:
   "INPUT MAPPING DB"."P-601 ON" := "P-601 ON";
END_REGION

REGION Network 65: "P-801 A BACK WASH WAST FEED BACK"
   RUNG wire#powerrail
      Contact( "P-801 A BACK WASH WAST FEED BACK" )
      Coil( "INPUT MAPPING DB"."P-801 A BACK WASH WAST FEED BACK" )
   END_RUNG
   // the same network as SCL:
   "INPUT MAPPING DB"."P-801 A BACK WASH WAST FEED BACK" := "P-801 A BACK WASH WAST FEED BACK";
END_REGION

REGION Network 66: "P-801 B BACK WASH WAST FEED BACK"
   RUNG wire#powerrail
      Contact( "P-801 B BACK WASH WAST FEED BACK" )
      Coil( "INPUT MAPPING DB"."P-801 B BACK WASH WAST FEED BACK" )
   END_RUNG
   // the same network as SCL:
   "INPUT MAPPING DB"."P-801 B BACK WASH WAST FEED BACK" := "P-801 B BACK WASH WAST FEED BACK";
END_REGION

REGION Network 67: "SPARE(5)"
   RUNG wire#powerrail
      Contact( "SPARE(5)" )
      Coil( "INPUT MAPPING DB"."SPARE(5)" )
   END_RUNG
   // the same network as SCL:
   "INPUT MAPPING DB"."SPARE(5)" := "SPARE(5)";
END_REGION

REGION Network 68: "SPARE(6)"
   RUNG wire#powerrail
      Contact( "SPARE(6)" )
      Coil( "INPUT MAPPING DB"."SPARE(6)" )
   END_RUNG
   // the same network as SCL:
   "INPUT MAPPING DB"."SPARE(6)" := "SPARE(6)";
END_REGION

REGION Network 69: "SPARE(7)"
   RUNG wire#powerrail
      Contact( "SPARE(7)" )
      Coil( "INPUT MAPPING DB"."SPARE(7)" )
   END_RUNG
   // the same network as SCL:
   "INPUT MAPPING DB"."SPARE(7)" := "SPARE(7)";
END_REGION

REGION Network 70: "SPARE(8)"
   RUNG wire#powerrail
      Contact( "SPARE(8)" )
      Coil( "INPUT MAPPING DB"."SPARE(8)" )
   END_RUNG
   // the same network as SCL:
   "INPUT MAPPING DB"."SPARE(8)" := "SPARE(8)";
END_REGION

REGION Network 71: "SPARE(9)"
   RUNG wire#powerrail
      Contact( "SPARE(9)" )
      Coil( "INPUT MAPPING DB"."SPARE(9)" )
   END_RUNG
   // the same network as SCL:
   "INPUT MAPPING DB"."SPARE(9)" := "SPARE(9)";
END_REGION

REGION Network 72: "SPARE(10)"
   RUNG wire#powerrail
      Contact( "SPARE(10)" )
      Coil( "INPUT MAPPING DB"."SPARE(10)" )
   END_RUNG
   // the same network as SCL:
   "INPUT MAPPING DB"."SPARE(10)" := "SPARE(10)";
END_REGION

REGION Network 73: "ABFV 501 OPEN FEED BACK"
   RUNG wire#powerrail
      Contact( "ABFV 501 OPEN FEED BACK" )
      Coil( "INPUT MAPPING DB"."ABFV 501 OPEN FEED BACK" )
   END_RUNG
   // the same network as SCL:
   "INPUT MAPPING DB"."ABFV 501 OPEN FEED BACK" := "ABFV 501 OPEN FEED BACK";
END_REGION

REGION Network 74: "ABFV 501 CLOSE FEED BACK"
   RUNG wire#powerrail
      Contact( "ABFV 501 CLOSE FEED BACK" )
      Coil( "INPUT MAPPING DB"."ABFV 501 CLOSE FEED BACK" )
   END_RUNG
   // the same network as SCL:
   "INPUT MAPPING DB"."ABFV 501 CLOSE FEED BACK" := "ABFV 501 CLOSE FEED BACK";
END_REGION

REGION Network 75: "ABFV 502 OPEN FEED BACK"
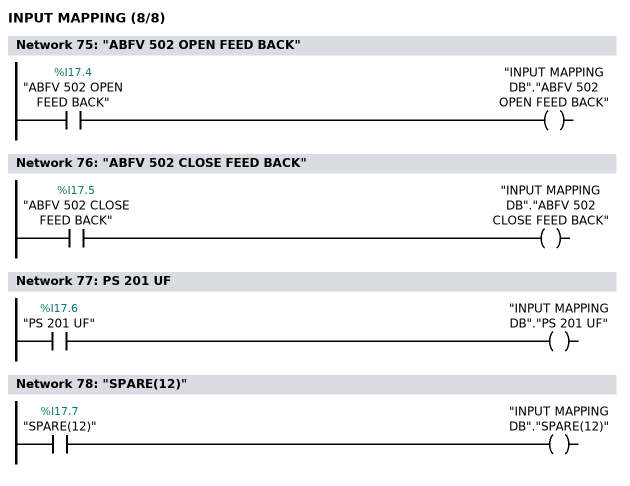
   RUNG wire#powerrail
      Contact( "ABFV 502 OPEN FEED BACK" )
      Coil( "INPUT MAPPING DB"."ABFV 502 OPEN FEED BACK" )
   END_RUNG
   // the same network as SCL:
   "INPUT MAPPING DB"."ABFV 502 OPEN FEED BACK" := "ABFV 502 OPEN FEED BACK";
END_REGION

REGION Network 76: "ABFV 502 CLOSE FEED BACK"
   RUNG wire#powerrail
      Contact( "ABFV 502 CLOSE FEED BACK" )
      Coil( "INPUT MAPPING DB"."ABFV 502 CLOSE FEED BACK" )
   END_RUNG
   // the same network as SCL:
   "INPUT MAPPING DB"."ABFV 502 CLOSE FEED BACK" := "ABFV 502 CLOSE FEED BACK";
END_REGION

REGION Network 77: PS 201 UF
   RUNG wire#powerrail
      Contact( "PS 201 UF" )
      Coil( "INPUT MAPPING DB"."PS 201 UF" )
   END_RUNG
   // the same network as SCL:
   "INPUT MAPPING DB"."PS 201 UF" := "PS 201 UF";
END_REGION

REGION Network 78: "SPARE(12)"
   RUNG wire#powerrail
      Contact( "SPARE(12)" )
      Coil( "INPUT MAPPING DB"."SPARE(12)" )
   END_RUNG
   // the same network as SCL:
   "INPUT MAPPING DB"."SPARE(12)" := "SPARE(12)";
END_REGION
END_FUNCTION

FUNCTION "OUTPUT MAPPING" : Void   // FC2, LAD
{ S7_Optimized_Access := 'TRUE' }
// stored: SetENOAutomatically false
BEGIN

REGION Network 1: "HOOTER RESET"
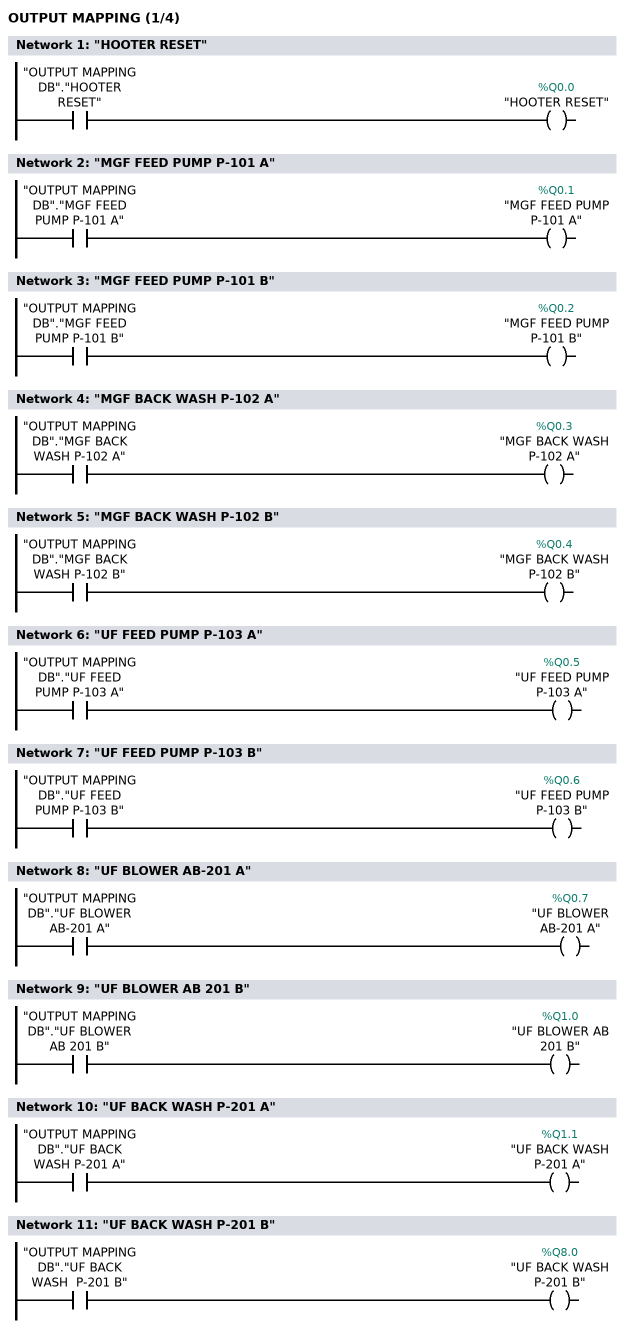
   RUNG wire#powerrail
      Contact( "OUTPUT MAPPING DB"."HOOTER RESET" )
      Coil( "HOOTER RESET" )
   END_RUNG
   // the same network as SCL:
   "HOOTER RESET" := "OUTPUT MAPPING DB"."HOOTER RESET";
END_REGION

REGION Network 2: "MGF FEED PUMP P-101 A"
   RUNG wire#powerrail
      Contact( "OUTPUT MAPPING DB"."MGF FEED PUMP P-101 A" )
      Coil( "MGF FEED PUMP P-101 A" )
   END_RUNG
   // the same network as SCL:
   "MGF FEED PUMP P-101 A" := "OUTPUT MAPPING DB"."MGF FEED PUMP P-101 A";
END_REGION

REGION Network 3: "MGF FEED PUMP P-101 B"
   RUNG wire#powerrail
      Contact( "OUTPUT MAPPING DB"."MGF FEED PUMP P-101 B" )
      Coil( "MGF FEED PUMP P-101 B" )
   END_RUNG
   // the same network as SCL:
   "MGF FEED PUMP P-101 B" := "OUTPUT MAPPING DB"."MGF FEED PUMP P-101 B";
END_REGION

REGION Network 4: "MGF BACK WASH P-102 A"
   RUNG wire#powerrail
      Contact( "OUTPUT MAPPING DB"."MGF BACK WASH P-102 A" )
      Coil( "MGF BACK WASH P-102 A" )
   END_RUNG
   // the same network as SCL:
   "MGF BACK WASH P-102 A" := "OUTPUT MAPPING DB"."MGF BACK WASH P-102 A";
END_REGION

REGION Network 5: "MGF BACK WASH P-102 B"
   RUNG wire#powerrail
      Contact( "OUTPUT MAPPING DB"."MGF BACK WASH P-102 B" )
      Coil( "MGF BACK WASH P-102 B" )
   END_RUNG
   // the same network as SCL:
   "MGF BACK WASH P-102 B" := "OUTPUT MAPPING DB"."MGF BACK WASH P-102 B";
END_REGION

REGION Network 6: "UF FEED PUMP P-103 A"
   RUNG wire#powerrail
      Contact( "OUTPUT MAPPING DB"."UF FEED PUMP P-103 A" )
      Coil( "UF FEED PUMP P-103 A" )
   END_RUNG
   // the same network as SCL:
   "UF FEED PUMP P-103 A" := "OUTPUT MAPPING DB"."UF FEED PUMP P-103 A";
END_REGION

REGION Network 7: "UF FEED PUMP P-103 B"
   RUNG wire#powerrail
      Contact( "OUTPUT MAPPING DB"."UF FEED PUMP P-103 B" )
      Coil( "UF FEED PUMP P-103 B" )
   END_RUNG
   // the same network as SCL:
   "UF FEED PUMP P-103 B" := "OUTPUT MAPPING DB"."UF FEED PUMP P-103 B";
END_REGION

REGION Network 8: "UF BLOWER AB-201 A"
   RUNG wire#powerrail
      Contact( "OUTPUT MAPPING DB"."UF BLOWER AB-201 A" )
      Coil( "UF BLOWER AB-201 A" )
   END_RUNG
   // the same network as SCL:
   "UF BLOWER AB-201 A" := "OUTPUT MAPPING DB"."UF BLOWER AB-201 A";
END_REGION

REGION Network 9: "UF BLOWER AB 201 B"
   RUNG wire#powerrail
      Contact( "OUTPUT MAPPING DB"."UF BLOWER AB 201 B" )
      Coil( "UF BLOWER AB 201 B" )
   END_RUNG
   // the same network as SCL:
   "UF BLOWER AB 201 B" := "OUTPUT MAPPING DB"."UF BLOWER AB 201 B";
END_REGION

REGION Network 10: "UF BACK WASH P-201 A"
   RUNG wire#powerrail
      Contact( "OUTPUT MAPPING DB"."UF BACK WASH P-201 A" )
      Coil( "UF BACK WASH P-201 A" )
   END_RUNG
   // the same network as SCL:
   "UF BACK WASH P-201 A" := "OUTPUT MAPPING DB"."UF BACK WASH P-201 A";
END_REGION

REGION Network 11: "UF BACK WASH P-201 B"
   RUNG wire#powerrail
      Contact( "OUTPUT MAPPING DB"."UF BACK WASH  P-201 B" )
      Coil( "UF BACK WASH  P-201 B" )
   END_RUNG
   // the same network as SCL:
   "UF BACK WASH  P-201 B" := "OUTPUT MAPPING DB"."UF BACK WASH  P-201 B";
END_REGION

REGION Network 12: "DM FEED PUMP P-502 A"
